  MoveL 4024 to (-41.13, 53.64, 69.25) mm, rotated rx -180 ry 0 rz 180 deg; joints [-165.068, 60.327, -74.122, 164.646, 76.68, 3.62]
  Call Extruder(59.42806)
  MoveL 4025 to (-41.09, 53.05, 69.25) mm, rotated rx -180 ry 0 rz -180 deg; joints [-165.222, 60.313, -74.132, 164.802, 76.647, 3.59]
  MoveL 4026 to (-41.09, 53.05, 69.25) mm, rotated rx -180 ry 0 rz -180 deg; joints [-165.222, 60.313, -74.132, 164.802, 76.647, 3.59]
  Call Extruder(59.67430)
  MoveL 4027 to (-41.04, 52.56, 69.25) mm, rotated rx -180 ry 0 rz -180 deg; joints [-165.349, 60.302, -74.14, 164.93, 76.62, 3.565]
  MoveL 4028 to (-41.04, 52.56, 69.25) mm, rotated rx -180 ry 0 rz -180 deg; joints [-165.349, 60.302, -74.14, 164.93, 76.62, 3.565]
  Call Extruder(59.87100)
  MoveL 4029 to (-40.99, 52.17, 69.25) mm, rotated rx 180 ry 0 rz 180 deg; joints [-165.449, 60.292, -74.147, 165.032, 76.597, 3.546]
  MoveL 4030 to (-40.99, 52.17, 69.25) mm, rotated rx 180 ry 0 rz 180 deg; joints [-165.449, 60.292, -74.147, 165.032, 76.597, 3.546]
  Call Extruder(60.06858)
  MoveL 4031 to (-40.95, 51.78, 69.25) mm, rotated rx -180 ry 0 rz -180 deg; joints [-165.549, 60.282, -74.154, 165.134, 76.575, 3.527]
  MoveL 4032 to (-40.95, 51.78, 69.25) mm, rotated rx -180 ry 0 rz -180 deg; joints [-165.549, 60.282, -74.154, 165.134, 76.575, 3.527]
  Call Extruder(60.26702)
  MoveL 4033 to (-40.9, 51.4, 69.25) mm, rotated rx 180 ry 0 rz -180 deg; joints [-165.65, 60.272, -74.162, 165.236, 76.552, 3.507]
  MoveL 4034 to (-40.9, 51.4, 69.25) mm, rotated rx 180 ry 0 rz -180 deg; joints [-165.65, 60.272, -74.162, 165.236, 76.552, 3.507]
  Call Extruder(60.46633)
  MoveL 4035 to (-40.86, 51.01, 69.25) mm, rotated rx -180 ry 0 rz -180 deg; joints [-165.751, 60.262, -74.169, 165.339, 76.53, 3.488]
  MoveL 4036 to (-40.86, 51.01, 69.25) mm, rotated rx -180 ry 0 rz -180 deg; joints [-165.751, 60.262, -74.169, 165.339, 76.53, 3.488]
  Call Extruder(60.62514)
  MoveL 4037 to (-40.81, 50.7, 69.25) mm, rotated rx 180 ry 0 rz -180 deg; joints [-165.829, 60.254, -74.175, 165.419, 76.511, 3.472]
  MoveL 4038 to (-40.81, 50.7, 69.25) mm, rotated rx 180 ry 0 rz -180 deg; joints [-165.829, 60.254, -74.175, 165.419, 76.511, 3.472]
  Call Extruder(60.78469)
  MoveL 4039 to (-40.76, 50.4, 69.25) mm, rotated rx -180 ry 0 rz -180 deg; joints [-165.908, 60.245, -74.181, 165.499, 76.492, 3.457]
  MoveL 4040 to (-40.76, 50.4, 69.25) mm, rotated rx -180 ry 0 rz -180 deg; joints [-165.908, 60.245, -74.181, 165.499, 76.492, 3.457]
  Call Extruder(60.94496)
  MoveL 4041 to (-40.71, 50.09, 69.25) mm, rotated rx -180 ry 0 rz -180 deg; joints [-165.987, 60.237, -74.187, 165.578, 76.473, 3.442]
  MoveL 4042 to (-40.71, 50.09, 69.25) mm, rotated rx -180 ry 0 rz -180 deg; joints [-165.987, 60.237, -74.187, 165.578, 76.473, 3.442]
  Call Extruder(61.10596)
  MoveL 4043 to (-40.66, 49.79, 69.25) mm, rotated rx 180 ry 0 rz 180 deg; joints [-166.066, 60.228, -74.193, 165.659, 76.454, 3.427]
  MoveL 4044 to (-40.66, 49.79, 69.25) mm, rotated rx 180 ry 0 rz 180 deg; joints [-166.066, 60.228, -74.193, 165.659, 76.454, 3.427]
  Call Extruder(61.26769)
  MoveL 4045 to (-40.61, 49.48, 69.25) mm, rotated rx 180 ry 0 rz 180 deg; joints [-166.145, 60.22, -74.199, 165.739, 76.435, 3.412]
  MoveL 4046 to (-40.61, 49.48, 69.25) mm, rotated rx 180 ry 0 rz 180 deg; joints [-166.145, 60.22, -74.199, 165.739, 76.435, 3.412]
  Call Extruder(61.43014)
  MoveL 4047 to (-40.57, 49.17, 69.25) mm, rotated rx -180 ry 0 rz -180 deg; joints [-166.224, 60.211, -74.205, 165.819, 76.417, 3.396]
  MoveL 4048 to (-40.57, 49.17, 69.25) mm, rotated rx -180 ry 0 rz -180 deg; joints [-166.224, 60.211, -74.205, 165.819, 76.417, 3.396]
  Call Extruder(61.56407)
  MoveL 4049 to (-40.52, 48.93, 69.25) mm, rotated rx -180 ry 0 rz -180 deg; joints [-166.288, 60.204, -74.21, 165.884, 76.4, 3.384]
  MoveL 4050 to (-40.52, 48.93, 69.25) mm, rotated rx -180 ry 0 rz -180 deg; joints [-166.288, 60.204, -74.21, 165.884, 76.4, 3.384]
  Call Extruder(61.69860)
  MoveL 4051 to (-40.47, 48.68, 69.25) mm, rotated rx -180 ry 0 rz 180 deg; joints [-166.352, 60.196, -74.216, 165.949, 76.384, 3.372]
  MoveL 4052 to (-40.47, 48.68, 69.25) mm, rotated rx -180 ry 0 rz 180 deg; joints [-166.352, 60.196, -74.216, 165.949, 76.384, 3.372]
  Call Extruder(61.83375)
  MoveL 4053 to (-40.42, 48.43, 69.25) mm, rotated rx -180 ry 0 rz -180 deg; joints [-166.416, 60.189, -74.221, 166.014, 76.368, 3.359]
  MoveL 4054 to (-40.42, 48.43, 69.25) mm, rotated rx -180 ry 0 rz -180 deg; joints [-166.416, 60.189, -74.221, 166.014, 76.368, 3.359]
  Call Extruder(61.96950)
  MoveL 4055 to (-40.37, 48.18, 69.25) mm, rotated rx -180 ry 0 rz -180 deg; joints [-166.48, 60.181, -74.226, 166.079, 76.352, 3.347]
  MoveL 4056 to (-40.37, 48.18, 69.25) mm, rotated rx -180 ry 0 rz -180 deg; joints [-166.48, 60.181, -74.226, 166.079, 76.352, 3.347]
  Call Extruder(62.10587)
  MoveL 4057 to (-40.32, 47.93, 69.25) mm, rotated rx -180 ry 0 rz 180 deg; joints [-166.544, 60.174, -74.231, 166.144, 76.336, 3.335]
  MoveL 4058 to (-40.32, 47.93, 69.25) mm, rotated rx -180 ry 0 rz 180 deg; joints [-166.544, 60.174, -74.231, 166.144, 76.336, 3.335]
  Call Extruder(62.24285)
  MoveL 4059 to (-40.27, 47.68, 69.25) mm, rotated rx -180 ry 0 rz -180 deg; joints [-166.608, 60.166, -74.237, 166.21, 76.32, 3.322]
  MoveL 4060 to (-40.27, 47.68, 69.25) mm, rotated rx -180 ry 0 rz -180 deg; joints [-166.608, 60.166, -74.237, 166.21, 76.32, 3.322]
  Call Extruder(62.38043)
  MoveL 4061 to (-40.22, 47.43, 69.25) mm, rotated rx -180 ry 0 rz 180 deg; joints [-166.673, 60.159, -74.242, 166.275, 76.304, 3.31]
  MoveL 4062 to (-40.22, 47.43, 69.25) mm, rotated rx -180 ry 0 rz 180 deg; joints [-166.673, 60.159, -74.242, 166.275, 76.304, 3.31]
  Call Extruder(62.49416)
  MoveL 4063 to (-40.17, 47.23, 69.25) mm, rotated rx -180 ry 0 rz 180 deg; joints [-166.725, 60.152, -74.246, 166.328, 76.29, 3.3]
  MoveL 4064 to (-40.17, 47.23, 69.25) mm, rotated rx -180 ry 0 rz 180 deg; joints [-166.725, 60.152, -74.246, 166.328, 76.29, 3.3]
  Call Extruder(62.60834)
  MoveL 4065 to (-40.13, 47.02, 69.25) mm, rotated rx -180 ry 0 rz 180 deg; joints [-166.778, 60.146, -74.251, 166.382, 76.276, 3.289]
  MoveL 4066 to (-40.13, 47.02, 69.25) mm, rotated rx -180 ry 0 rz 180 deg; joints [-166.778, 60.146, -74.251, 166.382, 76.276, 3.289]
  Call Extruder(62.72297)
  MoveL 4067 to (-40.08, 46.82, 69.25) mm, rotated rx 180 ry 0 rz -180 deg; joints [-166.83, 60.14, -74.255, 166.435, 76.263, 3.279]
  MoveL 4068 to (-40.08, 46.82, 69.25) mm, rotated rx 180 ry 0 rz -180 deg; joints [-166.83, 60.14, -74.255, 166.435, 76.263, 3.279]
  Call Extruder(62.83806)
  MoveL 4069 to (-40.04, 46.61, 69.25) mm, rotated rx -180 ry 0 rz -180 deg; joints [-166.883, 60.133, -74.26, 166.489, 76.249, 3.269]
  MoveL 4070 to (-40.04, 46.61, 69.25) mm, rotated rx -180 ry 0 rz -180 deg; joints [-166.883, 60.133, -74.26, 166.489, 76.249, 3.269]
  Call Extruder(62.96029)
  MoveL 4071 to (-39.98, 46.4, 69.25) mm, rotated rx -180 ry 0 rz -180 deg; joints [-166.937, 60.126, -74.265, 166.544, 76.234, 3.259]
  MoveL 4072 to (-39.98, 46.4, 69.25) mm, rotated rx -180 ry 0 rz -180 deg; joints [-166.937, 60.126, -74.265, 166.544, 76.234, 3.259]
  Call Extruder(63.08996)
  MoveL 4073 to (-39.92, 46.18, 69.25) mm, rotated rx -180 ry 0 rz -180 deg; joints [-166.994, 60.118, -74.271, 166.601, 76.218, 3.248]
  MoveL 4074 to (-39.92, 46.18, 69.25) mm, rotated rx -180 ry 0 rz -180 deg; joints [-166.994, 60.118, -74.271, 166.601, 76.218, 3.248]
  Call Extruder(63.22019)
  MoveL 4075 to (-39.85, 45.95, 69.25) mm, rotated rx 180 ry 0 rz -180 deg; joints [-167.051, 60.11, -74.276, 166.659, 76.201, 3.238]
  MoveL 4076 to (-39.85, 45.95, 69.25) mm, rotated rx 180 ry 0 rz -180 deg; joints [-167.051, 60.11, -74.276, 166.659, 76.201, 3.238]
  Call Extruder(63.35098)
  MoveL 4077 to (-39.78, 45.73, 69.25) mm, rotated rx 180 ry 0 rz -180 deg; joints [-167.107, 60.101, -74.282, 166.716, 76.184, 3.227]
  MoveL 4078 to (-39.78, 45.73, 69.25) mm, rotated rx 180 ry 0 rz -180 deg; joints [-167.107, 60.101, -74.282, 166.716, 76.184, 3.227]
  Call Extruder(63.48234)
  MoveL 4079 to (-39.71, 45.5, 69.25) mm, rotated rx -180 ry 0 rz -180 deg; joints [-167.164, 60.093, -74.288, 166.774, 76.167, 3.216]
  MoveL 4080 to (-39.71, 45.5, 69.25) mm, rotated rx -180 ry 0 rz -180 deg; joints [-167.164, 60.093, -74.288, 166.774, 76.167, 3.216]
  Call Extruder(63.59424)
  MoveL 4081 to (-39.65, 45.32, 69.25) mm, rotated rx -180 ry 0 rz -180 deg; joints [-167.212, 60.086, -74.293, 166.822, 76.153, 3.207]
  MoveL 4082 to (-39.65, 45.32, 69.25) mm, rotated rx -180 ry 0 rz -180 deg; joints [-167.212, 60.086, -74.293, 166.822, 76.153, 3.207]
  Call Extruder(63.70659)
  MoveL 4083 to (-39.59, 45.13, 69.25) mm, rotated rx 180 ry 0 rz 180 deg; joints [-167.26, 60.079, -74.298, 166.871, 76.138, 3.198]
  MoveL 4084 to (-39.59, 45.13, 69.25) mm, rotated rx 180 ry 0 rz 180 deg; joints [-167.26, 60.079, -74.298, 166.871, 76.138, 3.198]
  Call Extruder(63.81938)
  MoveL 4085 to (-39.53, 44.94, 69.25) mm, rotated rx -180 ry 0 rz 180 deg; joints [-167.307, 60.072, -74.303, 166.919, 76.124, 3.19]
  MoveL 4086 to (-39.53, 44.94, 69.25) mm, rotated rx -180 ry 0 rz 180 deg; joints [-167.307, 60.072, -74.303, 166.919, 76.124, 3.19]
  Call Extruder(63.93261)
  MoveL 4087 to (-39.47, 44.75, 69.25) mm, rotated rx -180 ry 0 rz -180 deg; joints [-167.355, 60.065, -74.308, 166.967, 76.109, 3.181]
  MoveL 4088 to (-39.47, 44.75, 69.25) mm, rotated rx -180 ry 0 rz -180 deg; joints [-167.355, 60.065, -74.308, 166.967, 76.109, 3.181]
  Call Extruder(64.04629)
  MoveL 4089 to (-39.41, 44.56, 69.25) mm, rotated rx -180 ry 0 rz -180 deg; joints [-167.403, 60.057, -74.313, 167.016, 76.095, 3.172]
  MoveL 4090 to (-39.41, 44.56, 69.25) mm, rotated rx -180 ry 0 rz -180 deg; joints [-167.403, 60.057, -74.313, 167.016, 76.095, 3.172]
  Call Extruder(64.22825)
  MoveL 4091 to (-39.29, 44.27, 69.25) mm, rotated rx -180 ry 0 rz 180 deg; joints [-167.475, 60.045, -74.321, 167.089, 76.07, 3.159]
  MoveL 4092 to (-39.29, 44.27, 69.25) mm, rotated rx -180 ry 0 rz 180 deg; joints [-167.475, 60.045, -74.321, 167.089, 76.07, 3.159]
  Call Extruder(64.41097)
  MoveL 4093 to (-39.17, 43.98, 69.25) mm, rotated rx 180 ry 0 rz 180 deg; joints [-167.548, 60.032, -74.33, 167.163, 76.045, 3.146]
  MoveL 4094 to (-39.17, 43.98, 69.25) mm, rotated rx 180 ry 0 rz 180 deg; joints [-167.548, 60.032, -74.33, 167.163, 76.045, 3.146]
  Call Extruder(64.58138)
  MoveL 4095 to (-39.05, 43.71, 69.25) mm, rotated rx -180 ry 0 rz -180 deg; joints [-167.615, 60.02, -74.339, 167.231, 76.021, 3.134]
  MoveL 4096 to (-39.05, 43.71, 69.25) mm, rotated rx -180 ry 0 rz -180 deg; joints [-167.615, 60.02, -74.339, 167.231, 76.021, 3.134]
  Call Extruder(64.73937)
  MoveL 4097 to (-38.94, 43.46, 69.25) mm, rotated rx -180 ry 0 rz 180 deg; joints [-167.677, 60.008, -74.346, 167.294, 75.999, 3.122]
  MoveL 4098 to (-38.94, 43.46, 69.25) mm, rotated rx -180 ry 0 rz 180 deg; joints [-167.677, 60.008, -74.346, 167.294, 75.999, 3.122]
  Call Extruder(64.89795)
  MoveL 4099 to (-38.84, 43.21, 69.25) mm, rotated rx -180 ry 0 rz -180 deg; joints [-167.739, 59.997, -74.354, 167.357, 75.977, 3.111]
  MoveL 4100 to (-38.84, 43.21, 69.25) mm, rotated rx -180 ry 0 rz -180 deg; joints [-167.739, 59.997, -74.354, 167.357, 75.977, 3.111]
  Call Extruder(65.10412)
  MoveL 4101 to (-38.66, 42.91, 69.25) mm, rotated rx -180 ry 0 rz -180 deg; joints [-167.813, 59.981, -74.365, 167.431, 75.946, 3.099]
  MoveL 4102 to (-38.66, 42.91, 69.25) mm, rotated rx -180 ry 0 rz -180 deg; joints [-167.813, 59.981, -74.365, 167.431, 75.946, 3.099]
  Call Extruder(65.31106)
  MoveL 4103 to (-38.49, 42.6, 69.25) mm, rotated rx -180 ry 0 rz 180 deg; joints [-167.886, 59.964, -74.377, 167.505, 75.914, 3.087]
  MoveL 4104 to (-38.49, 42.6, 69.25) mm, rotated rx -180 ry 0 rz 180 deg; joints [-167.886, 59.964, -74.377, 167.505, 75.914, 3.087]
  Call Extruder(65.51879)
  MoveL 4105 to (-38.31, 42.3, 69.25) mm, rotated rx 180 ry 0 rz 180 deg; joints [-167.96, 59.947, -74.388, 167.579, 75.883, 3.075]
  MoveL 4106 to (-38.31, 42.3, 69.25) mm, rotated rx 180 ry 0 rz 180 deg; joints [-167.96, 59.947, -74.388, 167.579, 75.883, 3.075]
  Call Extruder(65.72729)
  MoveL 4107 to (-38.14, 41.99, 69.25) mm, rotated rx -180 ry 0 rz -180 deg; joints [-168.033, 59.93, -74.4, 167.653, 75.852, 3.063]
  MoveL 4108 to (-38.14, 41.99, 69.25) mm, rotated rx -180 ry 0 rz -180 deg; joints [-168.033, 59.93, -74.4, 167.653, 75.852, 3.063]
  Call Extruder(65.90684)
  MoveL 4109 to (-37.96, 41.75, 69.25) mm, rotated rx 180 ry 0 rz -180 deg; joints [-168.091, 59.914, -74.41, 167.711, 75.822, 3.054]
  MoveL 4110 to (-37.96, 41.75, 69.25) mm, rotated rx 180 ry 0 rz -180 deg; joints [-168.091, 59.914, -74.41, 167.711, 75.822, 3.054]
  Call Extruder(66.24028)
  MoveL 4111 to (-37.63, 41.3, 69.25) mm, rotated rx -180 ry 0 rz -180 deg; joints [-168.197, 59.885, -74.43, 167.818, 75.768, 3.038]
  MoveL 4112 to (-37.63, 41.3, 69.25) mm, rotated rx -180 ry 0 rz -180 deg; joints [-168.197, 59.885, -74.43, 167.818, 75.768, 3.038]
  Call Extruder(66.57490)
  MoveL 4113 to (-37.3, 40.85, 69.25) mm, rotated rx 180 ry 0 rz -180 deg; joints [-168.304, 59.855, -74.45, 167.925, 75.714, 3.022]
  Call Extruder(67.40283)
  MoveL 4114 to (-36.39, 39.81, 69.25) mm, rotated rx 180 ry 0 rz 180 deg; joints [-168.541, 59.776, -74.503, 168.163, 75.573, 2.989]
  Call Extruder(68.23074)
  MoveL 4115 to (-35.35, 38.9, 69.25) mm, rotated rx -180 ry 0 rz 180 deg; joints [-168.739, 59.69, -74.559, 168.359, 75.423, 2.968]
  Call Extruder(68.39804)
  MoveL 4116 to (-35.13, 38.73, 69.25) mm, rotated rx -180 ry 0 rz 180 deg; joints [-168.773, 59.671, -74.571, 168.392, 75.392, 2.966]
  MoveL 4117 to (-35.13, 38.73, 69.25) mm, rotated rx -180 ry 0 rz 180 deg; joints [-168.773, 59.671, -74.571, 168.392, 75.392, 2.966]
  Call Extruder(68.73147)
  MoveL 4118 to (-34.68, 38.41, 69.25) mm, rotated rx -180 ry 0 rz 180 deg; joints [-168.84, 59.635, -74.595, 168.459, 75.329, 2.961]
  MoveL 4119 to (-34.68, 38.41, 69.25) mm, rotated rx -180 ry 0 rz 180 deg; joints [-168.84, 59.635, -74.595, 168.459, 75.329, 2.961]
  Call Extruder(69.06371)
  MoveL 4120 to (-34.23, 38.08, 69.25) mm, rotated rx 180 ry 0 rz -180 deg; joints [-168.908, 59.598, -74.619, 168.526, 75.266, 2.955]
  MoveL 4121 to (-34.23, 38.08, 69.25) mm, rotated rx 180 ry 0 rz -180 deg; joints [-168.908, 59.598, -74.619, 168.526, 75.266, 2.955]
  Call Extruder(69.18141)
  MoveL 4122 to (-34.05, 37.98, 69.25) mm, rotated rx -180 ry 0 rz 180 deg; joints [-168.927, 59.584, -74.627, 168.544, 75.243, 2.955]
  MoveL 4123 to (-34.05, 37.98, 69.25) mm, rotated rx -180 ry 0 rz 180 deg; joints [-168.927, 59.584, -74.627, 168.544, 75.243, 2.955]
  Call Extruder(69.38913)
  MoveL 4124 to (-33.75, 37.8, 69.25) mm, rotated rx -180 ry 0 rz 180 deg; joints [-168.96, 59.56, -74.643, 168.576, 75.203, 2.954]
  MoveL 4125 to (-33.75, 37.8, 69.25) mm, rotated rx -180 ry 0 rz 180 deg; joints [-168.96, 59.56, -74.643, 168.576, 75.203, 2.954]
  Call Extruder(69.59607)
  MoveL 4126 to (-33.45, 37.63, 69.25) mm, rotated rx -180 ry 0 rz 180 deg; joints [-168.993, 59.536, -74.658, 168.609, 75.162, 2.954]
  MoveL 4127 to (-33.45, 37.63, 69.25) mm, rotated rx -180 ry 0 rz 180 deg; joints [-168.993, 59.536, -74.658, 168.609, 75.162, 2.954]
  Call Extruder(69.80224)
  MoveL 4128 to (-33.14, 37.45, 69.25) mm, rotated rx -180 ry 0 rz -180 deg; joints [-169.026, 59.512, -74.673, 168.641, 75.122, 2.953]
  MoveL 4129 to (-33.14, 37.45, 69.25) mm, rotated rx -180 ry 0 rz -180 deg; joints [-169.026, 59.512, -74.673, 168.641, 75.122, 2.953]
  Call Extruder(69.98392)
  MoveL 4130 to (-32.86, 37.31, 69.25) mm, rotated rx 180 ry 0 rz 180 deg; joints [-169.052, 59.49, -74.687, 168.665, 75.086, 2.953]
  MoveL 4131 to (-32.86, 37.31, 69.25) mm, rotated rx 180 ry 0 rz 180 deg; joints [-169.052, 59.49, -74.687, 168.665, 75.086, 2.953]
  Call Extruder(70.14192)
  MoveL 4132 to (-32.62, 37.2, 69.25) mm, rotated rx -180 ry 0 rz -180 deg; joints [-169.068, 59.47, -74.699, 168.681, 75.054, 2.955]
  MoveL 4133 to (-32.62, 37.2, 69.25) mm, rotated rx -180 ry 0 rz -180 deg; joints [-169.068, 59.47, -74.699, 168.681, 75.054, 2.955]
  Call Extruder(70.29931)
  MoveL 4134 to (-32.37, 37.1, 69.25) mm, rotated rx 180 ry 0 rz -180 deg; joints [-169.085, 59.451, -74.711, 168.697, 75.022, 2.957]
  MoveL 4135 to (-32.37, 37.1, 69.25) mm, rotated rx 180 ry 0 rz -180 deg; joints [-169.085, 59.451, -74.711, 168.697, 75.022, 2.957]
  Call Extruder(70.48203)
  MoveL 4136 to (-32.07, 36.97, 69.25) mm, rotated rx 180 ry 0 rz 180 deg; joints [-169.104, 59.428, -74.726, 168.714, 74.985, 2.96]
  MoveL 4137 to (-32.07, 36.97, 69.25) mm, rotated rx 180 ry 0 rz 180 deg; joints [-169.104, 59.428, -74.726, 168.714, 74.985, 2.96]
  Call Extruder(70.66398)
  MoveL 4138 to (-31.78, 36.85, 69.25) mm, rotated rx -180 ry 0 rz 180 deg; joints [-169.122, 59.406, -74.74, 168.731, 74.948, 2.962]
  MoveL 4139 to (-31.78, 36.85, 69.25) mm, rotated rx -180 ry 0 rz 180 deg; joints [-169.122, 59.406, -74.74, 168.731, 74.948, 2.962]
  Call Extruder(70.81131)
  MoveL 4140 to (-31.54, 36.76, 69.25) mm, rotated rx -180 ry 0 rz -180 deg; joints [-169.135, 59.387, -74.751, 168.743, 74.918, 2.965]
  MoveL 4141 to (-31.54, 36.76, 69.25) mm, rotated rx -180 ry 0 rz -180 deg; joints [-169.135, 59.387, -74.751, 168.743, 74.918, 2.965]
  Call Extruder(70.92455)
  MoveL 4142 to (-31.35, 36.7, 69.25) mm, rotated rx 180 ry 0 rz 180 deg; joints [-169.143, 59.373, -74.76, 168.749, 74.894, 2.968]
  MoveL 4143 to (-31.35, 36.7, 69.25) mm, rotated rx 180 ry 0 rz 180 deg; joints [-169.143, 59.373, -74.76, 168.749, 74.894, 2.968]
  Call Extruder(71.03734)
  MoveL 4144 to (-31.17, 36.64, 69.25) mm, rotated rx -180 ry 0 rz -180 deg; joints [-169.15, 59.358, -74.769, 168.755, 74.871, 2.97]
  MoveL 4145 to (-31.17, 36.64, 69.25) mm, rotated rx -180 ry 0 rz -180 deg; joints [-169.15, 59.358, -74.769, 168.755, 74.871, 2.97]
  Call Extruder(71.14968)
  MoveL 4146 to (-30.98, 36.58, 69.25) mm, rotated rx 180 ry 0 rz 180 deg; joints [-169.157, 59.344, -74.778, 168.762, 74.848, 2.973]
  MoveL 4147 to (-30.98, 36.58, 69.25) mm, rotated rx 180 ry 0 rz 180 deg; joints [-169.157, 59.344, -74.778, 168.762, 74.848, 2.973]
  Call Extruder(71.26159)
  MoveL 4148 to (-30.79, 36.52, 69.25) mm, rotated rx -180 ry 0 rz -180 deg; joints [-169.164, 59.329, -74.787, 168.768, 74.825, 2.976]
  MoveL 4149 to (-30.79, 36.52, 69.25) mm, rotated rx -180 ry 0 rz -180 deg; joints [-169.164, 59.329, -74.787, 168.768, 74.825, 2.976]
  Call Extruder(71.38299)
  MoveL 4150 to (-30.58, 36.45, 69.25) mm, rotated rx -180 ry 0 rz -180 deg; joints [-169.172, 59.313, -74.797, 168.774, 74.799, 2.979]
  MoveL 4151 to (-30.58, 36.45, 69.25) mm, rotated rx -180 ry 0 rz -180 deg; joints [-169.172, 59.313, -74.797, 168.774, 74.799, 2.979]
  Call Extruder(71.51378)
  MoveL 4152 to (-30.36, 36.38, 69.25) mm, rotated rx -180 ry 0 rz 180 deg; joints [-169.179, 59.296, -74.807, 168.78, 74.772, 2.983]
  MoveL 4153 to (-30.36, 36.38, 69.25) mm, rotated rx -180 ry 0 rz 180 deg; joints [-169.179, 59.296, -74.807, 168.78, 74.772, 2.983]
  Call Extruder(71.64400)
  MoveL 4154 to (-30.14, 36.32, 69.25) mm, rotated rx 180 ry 0 rz 180 deg; joints [-169.186, 59.279, -74.817, 168.786, 74.744, 2.986]
  MoveL 4155 to (-30.14, 36.32, 69.25) mm, rotated rx 180 ry 0 rz 180 deg; joints [-169.186, 59.279, -74.817, 168.786, 74.744, 2.986]
  Call Extruder(71.77367)
  MoveL 4156 to (-29.91, 36.25, 69.25) mm, rotated rx -180 ry 0 rz 180 deg; joints [-169.193, 59.262, -74.828, 168.792, 74.717, 2.99]
  MoveL 4157 to (-29.91, 36.25, 69.25) mm, rotated rx -180 ry 0 rz 180 deg; joints [-169.193, 59.262, -74.828, 168.792, 74.717, 2.99]
  Call Extruder(71.90276)
  MoveL 4158 to (-29.69, 36.18, 69.25) mm, rotated rx -180 ry 0 rz -180 deg; joints [-169.201, 59.245, -74.838, 168.798, 74.689, 2.993]
  MoveL 4159 to (-29.69, 36.18, 69.25) mm, rotated rx -180 ry 0 rz -180 deg; joints [-169.201, 59.245, -74.838, 168.798, 74.689, 2.993]
  Call Extruder(72.01784)
  MoveL 4160 to (-29.48, 36.14, 69.25) mm, rotated rx -180 ry 0 rz 180 deg; joints [-169.202, 59.229, -74.848, 168.799, 74.665, 2.998]
  MoveL 4161 to (-29.48, 36.14, 69.25) mm, rotated rx -180 ry 0 rz 180 deg; joints [-169.202, 59.229, -74.848, 168.799, 74.665, 2.998]
  Call Extruder(72.13246)
  MoveL 4162 to (-29.28, 36.09, 69.25) mm, rotated rx -180 ry 0 rz -180 deg; joints [-169.204, 59.214, -74.857, 168.799, 74.64, 3.002]
  MoveL 4163 to (-29.28, 36.09, 69.25) mm, rotated rx -180 ry 0 rz -180 deg; joints [-169.204, 59.214, -74.857, 168.799, 74.64, 3.002]
  Call Extruder(72.24663)
  MoveL 4164 to (-29.08, 36.05, 69.25) mm, rotated rx 180 ry 0 rz 180 deg; joints [-169.206, 59.198, -74.866, 168.799, 74.616, 3.007]
  MoveL 4165 to (-29.08, 36.05, 69.25) mm, rotated rx 180 ry 0 rz 180 deg; joints [-169.206, 59.198, -74.866, 168.799, 74.616, 3.007]
  Call Extruder(72.36034)
  MoveL 4166 to (-28.87, 36, 69.25) mm, rotated rx 180 ry 0 rz 180 deg; joints [-169.207, 59.183, -74.876, 168.8, 74.591, 3.012]
  MoveL 4167 to (-28.87, 36, 69.25) mm, rotated rx 180 ry 0 rz 180 deg; joints [-169.207, 59.183, -74.876, 168.8, 74.591, 3.012]
  Call Extruder(72.48576)
  MoveL 4168 to (-28.65, 35.96, 69.25) mm, rotated rx -180 ry 0 rz -180 deg; joints [-169.208, 59.165, -74.886, 168.8, 74.565, 3.017]
  MoveL 4169 to (-28.65, 35.96, 69.25) mm, rotated rx -180 ry 0 rz -180 deg; joints [-169.208, 59.165, -74.886, 168.8, 74.565, 3.017]
  Call Extruder(72.62274)
  MoveL 4170 to (-28.4, 35.91, 69.25) mm, rotated rx -180 ry 0 rz 180 deg; joints [-169.209, 59.146, -74.897, 168.799, 74.535, 3.023]
  MoveL 4171 to (-28.4, 35.91, 69.25) mm, rotated rx -180 ry 0 rz 180 deg; joints [-169.209, 59.146, -74.897, 168.799, 74.535, 3.023]
  Call Extruder(72.75911)
  MoveL 4172 to (-28.15, 35.86, 69.25) mm, rotated rx 180 ry 0 rz -180 deg; joints [-169.21, 59.128, -74.908, 168.797, 74.505, 3.029]
  MoveL 4173 to (-28.15, 35.86, 69.25) mm, rotated rx 180 ry 0 rz -180 deg; joints [-169.21, 59.128, -74.908, 168.797, 74.505, 3.029]
  Call Extruder(72.89487)
  MoveL 4174 to (-27.9, 35.81, 69.25) mm, rotated rx -180 ry 0 rz 180 deg; joints [-169.21, 59.109, -74.92, 168.797, 74.476, 3.035]
  MoveL 4175 to (-27.9, 35.81, 69.25) mm, rotated rx -180 ry 0 rz 180 deg; joints [-169.21, 59.109, -74.92, 168.797, 74.476, 3.035]
  Call Extruder(73.03001)
  MoveL 4176 to (-27.65, 35.76, 69.25) mm, rotated rx -180 ry 0 rz 180 deg; joints [-169.211, 59.09, -74.931, 168.795, 74.446, 3.04]
  MoveL 4177 to (-27.65, 35.76, 69.25) mm, rotated rx -180 ry 0 rz 180 deg; joints [-169.211, 59.09, -74.931, 168.795, 74.446, 3.04]
  Call Extruder(73.16455)
  MoveL 4178 to (-27.4, 35.71, 69.25) mm, rotated rx 180 ry 0 rz -180 deg; joints [-169.212, 59.071, -74.942, 168.795, 74.417, 3.046]
  MoveL 4179 to (-27.4, 35.71, 69.25) mm, rotated rx 180 ry 0 rz -180 deg; joints [-169.212, 59.071, -74.942, 168.795, 74.417, 3.046]
  Call Extruder(73.29848)
  MoveL 4180 to (-27.15, 35.66, 69.25) mm, rotated rx 180 ry 0 rz 180 deg; joints [-169.212, 59.052, -74.953, 168.793, 74.387, 3.052]
  MoveL 4181 to (-27.15, 35.66, 69.25) mm, rotated rx 180 ry 0 rz 180 deg; joints [-169.212, 59.052, -74.953, 168.793, 74.387, 3.052]
  Call Extruder(73.44634)
  MoveL 4182 to (-26.87, 35.61, 69.25) mm, rotated rx -180 ry 0 rz 180 deg; joints [-169.211, 59.031, -74.965, 168.791, 74.354, 3.059]
  MoveL 4183 to (-26.87, 35.61, 69.25) mm, rotated rx -180 ry 0 rz 180 deg; joints [-169.211, 59.031, -74.965, 168.791, 74.354, 3.059]
  Call Extruder(73.60807)
  MoveL 4184 to (-26.57, 35.56, 69.25) mm, rotated rx -180 ry 0 rz -180 deg; joints [-169.208, 59.007, -74.979, 168.786, 74.318, 3.068]
  MoveL 4185 to (-26.57, 35.56, 69.25) mm, rotated rx -180 ry 0 rz -180 deg; joints [-169.208, 59.007, -74.979, 168.786, 74.318, 3.068]
  Call Extruder(73.76908)
  MoveL 4186 to (-26.26, 35.51, 69.25) mm, rotated rx 180 ry 0 rz 180 deg; joints [-169.205, 58.984, -74.992, 168.78, 74.283, 3.076]
  MoveL 4187 to (-26.26, 35.51, 69.25) mm, rotated rx 180 ry 0 rz 180 deg; joints [-169.205, 58.984, -74.992, 168.78, 74.283, 3.076]
  Call Extruder(73.92935)
  MoveL 4188 to (-25.96, 35.47, 69.25) mm, rotated rx -180 ry 0 rz -180 deg; joints [-169.202, 58.961, -75.006, 168.776, 74.247, 3.084]
  MoveL 4189 to (-25.96, 35.47, 69.25) mm, rotated rx -180 ry 0 rz -180 deg; joints [-169.202, 58.961, -75.006, 168.776, 74.247, 3.084]
  Call Extruder(74.08890)
  MoveL 4190 to (-25.65, 35.42, 69.25) mm, rotated rx -180 ry 0 rz 180 deg; joints [-169.199, 58.938, -75.019, 168.77, 74.211, 3.092]
  MoveL 4191 to (-25.65, 35.42, 69.25) mm, rotated rx -180 ry 0 rz 180 deg; joints [-169.199, 58.938, -75.019, 168.77, 74.211, 3.092]
  Call Extruder(74.24773)
  MoveL 4192 to (-25.34, 35.37, 69.25) mm, rotated rx -180 ry 0 rz 180 deg; joints [-169.196, 58.914, -75.032, 168.765, 74.175, 3.1]
  MoveL 4193 to (-25.34, 35.37, 69.25) mm, rotated rx -180 ry 0 rz 180 deg; joints [-169.196, 58.914, -75.032, 168.765, 74.175, 3.1]
  Call Extruder(74.42640)
  MoveL 4194 to (-25, 35.32, 69.25) mm, rotated rx 180 ry 0 rz 180 deg; joints [-169.191, 58.888, -75.047, 168.757, 74.135, 3.11]
  MoveL 4195 to (-25, 35.32, 69.25) mm, rotated rx 180 ry 0 rz 180 deg; joints [-169.191, 58.888, -75.047, 168.757, 74.135, 3.11]
  Call Extruder(74.62484)
  MoveL 4196 to (-24.61, 35.28, 69.25) mm, rotated rx -180 ry 0 rz 180 deg; joints [-169.182, 58.859, -75.064, 168.746, 74.09, 3.122]
  MoveL 4197 to (-24.61, 35.28, 69.25) mm, rotated rx -180 ry 0 rz 180 deg; joints [-169.182, 58.859, -75.064, 168.746, 74.09, 3.122]
  Call Extruder(74.82241)
  MoveL 4198 to (-24.22, 35.23, 69.25) mm, rotated rx 180 ry 0 rz 180 deg; joints [-169.174, 58.829, -75.081, 168.735, 74.046, 3.134]
  MoveL 4199 to (-24.22, 35.23, 69.25) mm, rotated rx 180 ry 0 rz 180 deg; joints [-169.174, 58.829, -75.081, 168.735, 74.046, 3.134]
  Call Extruder(75.01912)
  MoveL 4200 to (-23.83, 35.18, 69.25) mm, rotated rx -180 ry 0 rz -180 deg; joints [-169.166, 58.8, -75.097, 168.723, 74.001, 3.146]
  MoveL 4201 to (-23.83, 35.18, 69.25) mm, rotated rx -180 ry 0 rz -180 deg; joints [-169.166, 58.8, -75.097, 168.723, 74.001, 3.146]
  Call Extruder(75.21496)
  MoveL 4202 to (-23.45, 35.14, 69.25) mm, rotated rx 180 ry 0 rz -180 deg; joints [-169.157, 58.77, -75.114, 168.712, 73.956, 3.158]
  MoveL 4203 to (-23.45, 35.14, 69.25) mm, rotated rx 180 ry 0 rz -180 deg; joints [-169.157, 58.77, -75.114, 168.712, 73.956, 3.158]
  Call Extruder(75.51035)
  MoveL 4204 to (-22.86, 35.09, 69.25) mm, rotated rx -180 ry 0 rz 180 deg; joints [-169.137, 58.726, -75.139, 168.687, 73.889, 3.177]
  MoveL 4205 to (-22.86, 35.09, 69.25) mm, rotated rx -180 ry 0 rz 180 deg; joints [-169.137, 58.726, -75.139, 168.687, 73.889, 3.177]
  Call Extruder(75.80442)
  MoveL 4206 to (-22.27, 35.04, 69.25) mm, rotated rx 180 ry 0 rz 180 deg; joints [-169.117, 58.681, -75.163, 168.662, 73.823, 3.198]
  MoveL 4207 to (-22.27, 35.04, 69.25) mm, rotated rx 180 ry 0 rz 180 deg; joints [-169.117, 58.681, -75.163, 168.662, 73.823, 3.198]
  Call Extruder(76.09715)
  MoveL 4208 to (-21.68, 35, 69.25) mm, rotated rx -180 ry 0 rz 180 deg; joints [-169.096, 58.636, -75.188, 168.637, 73.756, 3.218]
  MoveL 4209 to (-21.68, 35, 69.25) mm, rotated rx -180 ry 0 rz 180 deg; joints [-169.096, 58.636, -75.188, 168.637, 73.756, 3.218]
  Call Extruder(76.67060)
  MoveL 4210 to (-20.52, 34.95, 69.25) mm, rotated rx -180 ry 0 rz -180 deg; joints [-169.042, 58.548, -75.235, 168.573, 73.626, 3.261]
  MoveL 4211 to (-20.52, 34.95, 69.25) mm, rotated rx -180 ry 0 rz -180 deg; joints [-169.042, 58.548, -75.235, 168.573, 73.626, 3.261]
  Call Extruder(77.38456)
  MoveL 4212 to (-19.06, 34.91, 69.25) mm, rotated rx -180 ry 0 rz 180 deg; joints [-168.967, 58.438, -75.294, 168.485, 73.464, 3.318]
  Call Extruder(194.23128)
  MoveL 4213 to (219.06, 34.91, 69.25) mm, rotated rx 180 ry 0 rz 180 deg; joints [-30.588, 47.996, -77.471, 34.176, 115.06, 16.045]
  Call Extruder(194.65984)
  MoveL 4214 to (219.94, 34.93, 69.25) mm, rotated rx 180 ry 0 rz 180 deg; joints [-30.233, 48.077, -77.472, 33.779, 115.092, 15.837]
  MoveL 4215 to (219.94, 34.93, 69.25) mm, rotated rx 180 ry 0 rz 180 deg; joints [-30.233, 48.077, -77.472, 33.779, 115.092, 15.837]
  Call Extruder(195.23329)
  MoveL 4216 to (221.1, 34.97, 69.25) mm, rotated rx -180 ry 0 rz 180 deg; joints [-29.789, 48.184, -77.474, 33.279, 115.124, 15.572]
  MoveL 4217 to (221.1, 34.97, 69.25) mm, rotated rx -180 ry 0 rz 180 deg; joints [-29.789, 48.184, -77.474, 33.279, 115.124, 15.572]
  Call Extruder(195.66760)
  MoveL 4218 to (221.97, 35.02, 69.25) mm, rotated rx 180 ry 0 rz 180 deg; joints [-29.47, 48.266, -77.476, 32.92, 115.142, 15.379]
  MoveL 4219 to (221.97, 35.02, 69.25) mm, rotated rx 180 ry 0 rz 180 deg; joints [-29.47, 48.266, -77.476, 32.92, 115.142, 15.379]
  Call Extruder(195.96166)
  MoveL 4220 to (222.56, 35.07, 69.25) mm, rotated rx -180 ry 0 rz 180 deg; joints [-29.272, 48.322, -77.476, 32.694, 115.148, 15.256]
  MoveL 4221 to (222.56, 35.07, 69.25) mm, rotated rx -180 ry 0 rz 180 deg; joints [-29.272, 48.322, -77.476, 32.694, 115.148, 15.256]
  Call Extruder(196.25705)
  MoveL 4222 to (223.15, 35.11, 69.25) mm, rotated rx -180 ry 0 rz -180 deg; joints [-29.075, 48.378, -77.477, 32.47, 115.153, 15.134]
  MoveL 4223 to (223.15, 35.11, 69.25) mm, rotated rx -180 ry 0 rz -180 deg; joints [-29.075, 48.378, -77.477, 32.47, 115.153, 15.134]
  Call Extruder(196.50328)
  MoveL 4224 to (223.64, 35.16, 69.25) mm, rotated rx -180 ry 0 rz 180 deg; joints [-28.92, 48.425, -77.477, 32.293, 115.154, 15.036]
  MoveL 4225 to (223.64, 35.16, 69.25) mm, rotated rx -180 ry 0 rz 180 deg; joints [-28.92, 48.425, -77.477, 32.293, 115.154, 15.036]
  Call Extruder(196.69999)
  MoveL 4226 to (224.03, 35.21, 69.25) mm, rotated rx -180 ry 0 rz 180 deg; joints [-28.804, 48.463, -77.478, 32.16, 115.152, 14.962]
  MoveL 4227 to (224.03, 35.21, 69.25) mm, rotated rx -180 ry 0 rz 180 deg; joints [-28.804, 48.463, -77.478, 32.16, 115.152, 14.962]
  Call Extruder(196.89757)
  MoveL 4228 to (224.42, 35.25, 69.25) mm, rotated rx 180 ry 0 rz 180 deg; joints [-28.69, 48.501, -77.478, 32.029, 115.15, 14.888]
  MoveL 4229 to (224.42, 35.25, 69.25) mm, rotated rx 180 ry 0 rz 180 deg; joints [-28.69, 48.501, -77.478, 32.029, 115.15, 14.888]
  Call Extruder(197.09601)
  MoveL 4230 to (224.8, 35.3, 69.25) mm, rotated rx -180 ry 0 rz 180 deg; joints [-28.577, 48.538, -77.478, 31.899, 115.147, 14.815]
  MoveL 4231 to (224.8, 35.3, 69.25) mm, rotated rx -180 ry 0 rz 180 deg; joints [-28.577, 48.538, -77.478, 31.899, 115.147, 14.815]
  Call Extruder(197.29532)
  MoveL 4232 to (225.19, 35.34, 69.25) mm, rotated rx -180 ry 0 rz 180 deg; joints [-28.465, 48.576, -77.478, 31.77, 115.144, 14.742]
  MoveL 4233 to (225.19, 35.34, 69.25) mm, rotated rx -180 ry 0 rz 180 deg; joints [-28.465, 48.576, -77.478, 31.77, 115.144, 14.742]
  Call Extruder(197.45414)
  MoveL 4234 to (225.5, 35.39, 69.25) mm, rotated rx -180 ry 0 rz 180 deg; joints [-28.385, 48.606, -77.478, 31.677, 115.138, 14.688]
  MoveL 4235 to (225.5, 35.39, 69.25) mm, rotated rx -180 ry 0 rz 180 deg; joints [-28.385, 48.606, -77.478, 31.677, 115.138, 14.688]
  Call Extruder(197.61369)
  MoveL 4236 to (225.8, 35.44, 69.25) mm, rotated rx 180 ry 0 rz 180 deg; joints [-28.307, 48.637, -77.478, 31.586, 115.132, 14.635]
  MoveL 4237 to (225.8, 35.44, 69.25) mm, rotated rx 180 ry 0 rz 180 deg; joints [-28.307, 48.637, -77.478, 31.586, 115.132, 14.635]
  Call Extruder(197.77397)
  MoveL 4238 to (226.11, 35.49, 69.25) mm, rotated rx 180 ry 0 rz 180 deg; joints [-28.228, 48.667, -77.478, 31.495, 115.126, 14.582]
  MoveL 4239 to (226.11, 35.49, 69.25) mm, rotated rx 180 ry 0 rz 180 deg; joints [-28.228, 48.667, -77.478, 31.495, 115.126, 14.582]
  Call Extruder(197.93497)
  MoveL 4240 to (226.41, 35.54, 69.25) mm, rotated rx -180 ry 0 rz 180 deg; joints [-28.151, 48.697, -77.478, 31.405, 115.12, 14.53]
  MoveL 4241 to (226.41, 35.54, 69.25) mm, rotated rx -180 ry 0 rz 180 deg; joints [-28.151, 48.697, -77.478, 31.405, 115.12, 14.53]
  Call Extruder(198.09670)
  MoveL 4242 to (226.72, 35.59, 69.25) mm, rotated rx -180 ry 0 rz 180 deg; joints [-28.074, 48.727, -77.478, 31.315, 115.113, 14.477]
  MoveL 4243 to (226.72, 35.59, 69.25) mm, rotated rx -180 ry 0 rz 180 deg; joints [-28.074, 48.727, -77.478, 31.315, 115.113, 14.477]
  Call Extruder(198.25916)
  MoveL 4244 to (227.02, 35.63, 69.25) mm, rotated rx -180 ry 0 rz 180 deg; joints [-27.998, 48.758, -77.478, 31.226, 115.106, 14.425]
  MoveL 4245 to (227.02, 35.63, 69.25) mm, rotated rx -180 ry 0 rz 180 deg; joints [-27.998, 48.758, -77.478, 31.226, 115.106, 14.425]
  Call Extruder(198.39309)
  MoveL 4246 to (227.27, 35.68, 69.25) mm, rotated rx -180 ry 0 rz 180 deg; joints [-27.942, 48.783, -77.478, 31.161, 115.098, 14.386]
  MoveL 4247 to (227.27, 35.68, 69.25) mm, rotated rx -180 ry 0 rz 180 deg; joints [-27.942, 48.783, -77.478, 31.161, 115.098, 14.386]
  Call Extruder(198.52763)
  MoveL 4248 to (227.52, 35.73, 69.25) mm, rotated rx -180 ry 0 rz 180 deg; joints [-27.888, 48.808, -77.478, 31.096, 115.09, 14.347]
  MoveL 4249 to (227.52, 35.73, 69.25) mm, rotated rx -180 ry 0 rz 180 deg; joints [-27.888, 48.808, -77.478, 31.096, 115.09, 14.347]
  Call Extruder(198.66277)
  MoveL 4250 to (227.77, 35.78, 69.25) mm, rotated rx -180 ry 0 rz 180 deg; joints [-27.834, 48.833, -77.478, 31.032, 115.082, 14.308]
  MoveL 4251 to (227.77, 35.78, 69.25) mm, rotated rx -180 ry 0 rz 180 deg; joints [-27.834, 48.833, -77.478, 31.032, 115.082, 14.308]
  Call Extruder(198.79853)
  MoveL 4252 to (228.02, 35.83, 69.25) mm, rotated rx -180 ry 0 rz 180 deg; joints [-27.78, 48.858, -77.478, 30.968, 115.074, 14.269]
  MoveL 4253 to (228.02, 35.83, 69.25) mm, rotated rx -180 ry 0 rz 180 deg; joints [-27.78, 48.858, -77.478, 30.968, 115.074, 14.269]
  Call Extruder(198.93490)
  MoveL 4254 to (228.27, 35.88, 69.25) mm, rotated rx -180 ry 0 rz -180 deg; joints [-27.726, 48.884, -77.477, 30.905, 115.065, 14.23]
  MoveL 4255 to (228.27, 35.88, 69.25) mm, rotated rx -180 ry 0 rz -180 deg; joints [-27.726, 48.884, -77.477, 30.905, 115.065, 14.23]
  Call Extruder(199.07188)
  MoveL 4256 to (228.52, 35.93, 69.25) mm, rotated rx -180 ry 0 rz 180 deg; joints [-27.673, 48.909, -77.477, 30.841, 115.056, 14.191]
  MoveL 4257 to (228.52, 35.93, 69.25) mm, rotated rx -180 ry 0 rz 180 deg; joints [-27.673, 48.909, -77.477, 30.841, 115.056, 14.191]
  Call Extruder(199.20947)
  MoveL 4258 to (228.77, 35.98, 69.25) mm, rotated rx 180 ry 0 rz 180 deg; joints [-27.62, 48.934, -77.477, 30.779, 115.047, 14.153]
  MoveL 4259 to (228.77, 35.98, 69.25) mm, rotated rx 180 ry 0 rz 180 deg; joints [-27.62, 48.934, -77.477, 30.779, 115.047, 14.153]
  Call Extruder(199.32318)
  MoveL 4260 to (228.97, 36.03, 69.25) mm, rotated rx -180 ry 0 rz 180 deg; joints [-27.579, 48.955, -77.477, 30.73, 115.039, 14.123]
  MoveL 4261 to (228.97, 36.03, 69.25) mm, rotated rx -180 ry 0 rz 180 deg; joints [-27.579, 48.955, -77.477, 30.73, 115.039, 14.123]
  Call Extruder(199.43735)
  MoveL 4262 to (229.18, 36.07, 69.25) mm, rotated rx -180 ry 0 rz -180 deg; joints [-27.539, 48.975, -77.477, 30.682, 115.031, 14.093]
  MoveL 4263 to (229.18, 36.07, 69.25) mm, rotated rx -180 ry 0 rz -180 deg; joints [-27.539, 48.975, -77.477, 30.682, 115.031, 14.093]
  Call Extruder(199.55198)
  MoveL 4264 to (229.38, 36.12, 69.25) mm, rotated rx 180 ry 0 rz 180 deg; joints [-27.499, 48.996, -77.476, 30.634, 115.023, 14.063]
  MoveL 4265 to (229.38, 36.12, 69.25) mm, rotated rx 180 ry 0 rz 180 deg; joints [-27.499, 48.996, -77.476, 30.634, 115.023, 14.063]
  Call Extruder(199.66705)
  MoveL 4266 to (229.59, 36.16, 69.25) mm, rotated rx 180 ry 0 rz 180 deg; joints [-27.458, 49.017, -77.476, 30.586, 115.015, 14.033]
  MoveL 4267 to (229.59, 36.16, 69.25) mm, rotated rx 180 ry 0 rz 180 deg; joints [-27.458, 49.017, -77.476, 30.586, 115.015, 14.033]
  Call Extruder(199.78928)
  MoveL 4268 to (229.8, 36.22, 69.25) mm, rotated rx -180 ry 0 rz 180 deg; joints [-27.423, 49.039, -77.476, 30.543, 115.004, 14.004]
  MoveL 4269 to (229.8, 36.22, 69.25) mm, rotated rx -180 ry 0 rz 180 deg; joints [-27.423, 49.039, -77.476, 30.543, 115.004, 14.004]
  Call Extruder(199.91895)
  MoveL 4270 to (230.02, 36.28, 69.25) mm, rotated rx -180 ry 0 rz 180 deg; joints [-27.392, 49.063, -77.475, 30.504, 114.991, 13.976]
  MoveL 4271 to (230.02, 36.28, 69.25) mm, rotated rx -180 ry 0 rz 180 deg; joints [-27.392, 49.063, -77.475, 30.504, 114.991, 13.976]
  Call Extruder(200.04918)
  MoveL 4272 to (230.25, 36.35, 69.25) mm, rotated rx -180 ry 0 rz 180 deg; joints [-27.361, 49.086, -77.475, 30.465, 114.977, 13.949]
  MoveL 4273 to (230.25, 36.35, 69.25) mm, rotated rx -180 ry 0 rz 180 deg; joints [-27.361, 49.086, -77.475, 30.465, 114.977, 13.949]
  Call Extruder(200.17998)
  MoveL 4274 to (230.47, 36.42, 69.25) mm, rotated rx 180 ry 0 rz 180 deg; joints [-27.33, 49.11, -77.475, 30.426, 114.964, 13.922]
  MoveL 4275 to (230.47, 36.42, 69.25) mm, rotated rx 180 ry 0 rz 180 deg; joints [-27.33, 49.11, -77.475, 30.426, 114.964, 13.922]
  Call Extruder(200.31134)
  MoveL 4276 to (230.69, 36.49, 69.25) mm, rotated rx -180 ry 0 rz 180 deg; joints [-27.299, 49.134, -77.474, 30.388, 114.951, 13.894]
  MoveL 4277 to (230.69, 36.49, 69.25) mm, rotated rx -180 ry 0 rz 180 deg; joints [-27.299, 49.134, -77.474, 30.388, 114.951, 13.894]
  Call Extruder(200.42676)
  MoveL 4278 to (230.89, 36.55, 69.25) mm, rotated rx 180 ry 0 rz 180 deg; joints [-27.275, 49.154, -77.474, 30.357, 114.938, 13.872]
  MoveL 4279 to (230.89, 36.55, 69.25) mm, rotated rx 180 ry 0 rz 180 deg; joints [-27.275, 49.154, -77.474, 30.357, 114.938, 13.872]
  Call Extruder(200.54265)
  MoveL 4280 to (231.08, 36.61, 69.25) mm, rotated rx -180 ry 0 rz 180 deg; joints [-27.252, 49.175, -77.474, 30.327, 114.926, 13.85]
  MoveL 4281 to (231.08, 36.61, 69.25) mm, rotated rx -180 ry 0 rz 180 deg; joints [-27.252, 49.175, -77.474, 30.327, 114.926, 13.85]
  Call Extruder(200.65547)
  MoveL 4282 to (231.27, 36.67, 69.25) mm, rotated rx -180 ry 0 rz 180 deg; joints [-27.229, 49.195, -77.473, 30.298, 114.914, 13.828]
  MoveL 4283 to (231.27, 36.67, 69.25) mm, rotated rx -180 ry 0 rz 180 deg; joints [-27.229, 49.195, -77.473, 30.298, 114.914, 13.828]
  Call Extruder(200.76517)
  MoveL 4284 to (231.46, 36.73, 69.25) mm, rotated rx -180 ry 0 rz 180 deg; joints [-27.207, 49.215, -77.473, 30.27, 114.902, 13.807]
  MoveL 4285 to (231.46, 36.73, 69.25) mm, rotated rx -180 ry 0 rz 180 deg; joints [-27.207, 49.215, -77.473, 30.27, 114.902, 13.807]
  Call Extruder(200.87528)
  MoveL 4286 to (231.64, 36.79, 69.25) mm, rotated rx -180 ry 0 rz 180 deg; joints [-27.185, 49.234, -77.472, 30.242, 114.89, 13.786]
  MoveL 4287 to (231.64, 36.79, 69.25) mm, rotated rx -180 ry 0 rz 180 deg; joints [-27.185, 49.234, -77.472, 30.242, 114.89, 13.786]
  Call Extruder(201.05724)
  MoveL 4288 to (231.93, 36.91, 69.25) mm, rotated rx -180 ry 0 rz -180 deg; joints [-27.167, 49.266, -77.472, 30.214, 114.866, 13.76]
  MoveL 4289 to (231.93, 36.91, 69.25) mm, rotated rx -180 ry 0 rz -180 deg; joints [-27.167, 49.266, -77.472, 30.214, 114.866, 13.76]
  Call Extruder(201.23996)
  MoveL 4290 to (232.22, 37.04, 69.25) mm, rotated rx 180 ry 0 rz 180 deg; joints [-27.149, 49.299, -77.471, 30.187, 114.842, 13.733]
  MoveL 4291 to (232.22, 37.04, 69.25) mm, rotated rx 180 ry 0 rz 180 deg; joints [-27.149, 49.299, -77.471, 30.187, 114.842, 13.733]
  Call Extruder(201.41037)
  MoveL 4292 to (232.49, 37.15, 69.25) mm, rotated rx 180 ry 0 rz -180 deg; joints [-27.133, 49.328, -77.47, 30.164, 114.819, 13.709]
  MoveL 4293 to (232.49, 37.15, 69.25) mm, rotated rx 180 ry 0 rz -180 deg; joints [-27.133, 49.328, -77.47, 30.164, 114.819, 13.709]
  Call Extruder(201.56837)
  MoveL 4294 to (232.74, 37.26, 69.25) mm, rotated rx 180 ry 0 rz 180 deg; joints [-27.121, 49.356, -77.47, 30.143, 114.797, 13.688]
  MoveL 4295 to (232.74, 37.26, 69.25) mm, rotated rx 180 ry 0 rz 180 deg; joints [-27.121, 49.356, -77.47, 30.143, 114.797, 13.688]
  Call Extruder(201.72697)
  MoveL 4296 to (232.99, 37.36, 69.25) mm, rotated rx -180 ry 0 rz 180 deg; joints [-27.108, 49.384, -77.469, 30.123, 114.776, 13.666]
  MoveL 4297 to (232.99, 37.36, 69.25) mm, rotated rx -180 ry 0 rz 180 deg; joints [-27.108, 49.384, -77.469, 30.123, 114.776, 13.666]
  Call Extruder(201.93314)
  MoveL 4298 to (233.29, 37.54, 69.25) mm, rotated rx -180 ry 0 rz 180 deg; joints [-27.12, 49.42, -77.468, 30.127, 114.741, 13.651]
  MoveL 4299 to (233.29, 37.54, 69.25) mm, rotated rx -180 ry 0 rz 180 deg; joints [-27.12, 49.42, -77.468, 30.127, 114.741, 13.651]
  Call Extruder(202.14008)
  MoveL 4300 to (233.6, 37.71, 69.25) mm, rotated rx -180 ry 0 rz -180 deg; joints [-27.132, 49.455, -77.467, 30.132, 114.706, 13.637]
  MoveL 4301 to (233.6, 37.71, 69.25) mm, rotated rx -180 ry 0 rz -180 deg; joints [-27.132, 49.455, -77.467, 30.132, 114.706, 13.637]
  Call Extruder(202.34781)
  MoveL 4302 to (233.9, 37.89, 69.25) mm, rotated rx -180 ry 0 rz 180 deg; joints [-27.144, 49.491, -77.466, 30.136, 114.672, 13.622]
  MoveL 4303 to (233.9, 37.89, 69.25) mm, rotated rx -180 ry 0 rz 180 deg; joints [-27.144, 49.491, -77.466, 30.136, 114.672, 13.622]
  Call Extruder(202.55631)
  MoveL 4304 to (234.21, 38.07, 69.25) mm, rotated rx 180 ry 0 rz -180 deg; joints [-27.156, 49.527, -77.465, 30.141, 114.637, 13.607]
  MoveL 4305 to (234.21, 38.07, 69.25) mm, rotated rx 180 ry 0 rz -180 deg; joints [-27.156, 49.527, -77.465, 30.141, 114.637, 13.607]
  Call Extruder(202.73585)
  MoveL 4306 to (234.45, 38.24, 69.25) mm, rotated rx -180 ry 0 rz 180 deg; joints [-27.187, 49.557, -77.464, 30.166, 114.603, 13.603]
  MoveL 4307 to (234.45, 38.24, 69.25) mm, rotated rx -180 ry 0 rz 180 deg; joints [-27.187, 49.557, -77.464, 30.166, 114.603, 13.603]
  Call Extruder(203.06927)
  MoveL 4308 to (234.9, 38.57, 69.25) mm, rotated rx -180 ry 0 rz 180 deg; joints [-27.245, 49.613, -77.462, 30.215, 114.539, 13.597]
  MoveL 4309 to (234.9, 38.57, 69.25) mm, rotated rx -180 ry 0 rz 180 deg; joints [-27.245, 49.613, -77.462, 30.215, 114.539, 13.597]
  Call Extruder(203.40387)
  MoveL 4310 to (235.35, 38.9, 69.25) mm, rotated rx 180 ry 0 rz 180 deg; joints [-27.302, 49.669, -77.46, 30.263, 114.475, 13.59]
  Call Extruder(204.23182)
  MoveL 4311 to (236.39, 39.81, 69.25) mm, rotated rx -180 ry 0 rz 180 deg; joints [-27.525, 49.805, -77.455, 30.468, 114.301, 13.61]
  Call Extruder(205.05976)
  MoveL 4312 to (237.3, 40.85, 69.25) mm, rotated rx -180 ry 0 rz 180 deg; joints [-27.851, 49.936, -77.449, 30.785, 114.107, 13.676]
  Call Extruder(205.22706)
  MoveL 4313 to (237.47, 41.07, 69.25) mm, rotated rx 180 ry 0 rz -180 deg; joints [-27.932, 49.961, -77.448, 30.865, 114.065, 13.696]
  MoveL 4314 to (237.47, 41.07, 69.25) mm, rotated rx 180 ry 0 rz -180 deg; joints [-27.932, 49.961, -77.448, 30.865, 114.065, 13.696]
  Call Extruder(205.56048)
  MoveL 4315 to (237.79, 41.52, 69.25) mm, rotated rx -180 ry 0 rz 180 deg; joints [-28.091, 50.012, -77.445, 31.022, 113.982, 13.735]
  MoveL 4316 to (237.79, 41.52, 69.25) mm, rotated rx -180 ry 0 rz 180 deg; joints [-28.091, 50.012, -77.445, 31.022, 113.982, 13.735]
  Call Extruder(205.89270)
  MoveL 4317 to (238.12, 41.98, 69.25) mm, rotated rx -180 ry 0 rz -180 deg; joints [-28.249, 50.062, -77.443, 31.177, 113.899, 13.773]
  MoveL 4318 to (238.12, 41.98, 69.25) mm, rotated rx -180 ry 0 rz -180 deg; joints [-28.249, 50.062, -77.443, 31.177, 113.899, 13.773]
  Call Extruder(206.01040)
  MoveL 4319 to (238.22, 42.15, 69.25) mm, rotated rx 180 ry 0 rz 180 deg; joints [-28.315, 50.079, -77.442, 31.244, 113.868, 13.792]
  MoveL 4320 to (238.22, 42.15, 69.25) mm, rotated rx 180 ry 0 rz 180 deg; joints [-28.315, 50.079, -77.442, 31.244, 113.868, 13.792]
  Call Extruder(206.21813)
  MoveL 4321 to (238.4, 42.45, 69.25) mm, rotated rx -180 ry 0 rz 180 deg; joints [-28.434, 50.109, -77.44, 31.362, 113.812, 13.825]
  MoveL 4322 to (238.4, 42.45, 69.25) mm, rotated rx -180 ry 0 rz 180 deg; joints [-28.434, 50.109, -77.44, 31.362, 113.812, 13.825]
  Call Extruder(206.42507)
  MoveL 4323 to (238.57, 42.75, 69.25) mm, rotated rx 180 ry 0 rz 180 deg; joints [-28.552, 50.14, -77.439, 31.48, 113.757, 13.857]
  MoveL 4324 to (238.57, 42.75, 69.25) mm, rotated rx 180 ry 0 rz 180 deg; joints [-28.552, 50.14, -77.439, 31.48, 113.757, 13.857]
  Call Extruder(206.63124)
  MoveL 4325 to (238.75, 43.06, 69.25) mm, rotated rx 180 ry 0 rz 180 deg; joints [-28.669, 50.17, -77.437, 31.597, 113.702, 13.889]
  MoveL 4326 to (238.75, 43.06, 69.25) mm, rotated rx 180 ry 0 rz 180 deg; joints [-28.669, 50.17, -77.437, 31.597, 113.702, 13.889]
  Call Extruder(206.81293)
  MoveL 4327 to (238.89, 43.33, 69.25) mm, rotated rx -180 ry 0 rz 180 deg; joints [-28.78, 50.196, -77.436, 31.709, 113.652, 13.921]
  MoveL 4328 to (238.89, 43.33, 69.25) mm, rotated rx -180 ry 0 rz 180 deg; joints [-28.78, 50.196, -77.436, 31.709, 113.652, 13.921]
  Call Extruder(206.97094)
  MoveL 4329 to (239, 43.58, 69.25) mm, rotated rx 180 ry 0 rz 180 deg; joints [-28.886, 50.217, -77.434, 31.816, 113.607, 13.953]
  MoveL 4330 to (239, 43.58, 69.25) mm, rotated rx 180 ry 0 rz 180 deg; joints [-28.886, 50.217, -77.434, 31.816, 113.607, 13.953]
  Call Extruder(207.12835)
  MoveL 4331 to (239.11, 43.83, 69.25) mm, rotated rx -180 ry 0 rz 180 deg; joints [-28.991, 50.238, -77.433, 31.922, 113.562, 13.984]
  MoveL 4332 to (239.11, 43.83, 69.25) mm, rotated rx -180 ry 0 rz 180 deg; joints [-28.991, 50.238, -77.433, 31.922, 113.562, 13.984]
  Call Extruder(207.31106)
  MoveL 4333 to (239.23, 44.13, 69.25) mm, rotated rx -180 ry 0 rz -180 deg; joints [-29.116, 50.263, -77.432, 32.048, 113.51, 14.022]
  MoveL 4334 to (239.23, 44.13, 69.25) mm, rotated rx -180 ry 0 rz -180 deg; joints [-29.116, 50.263, -77.432, 32.048, 113.51, 14.022]
  Call Extruder(207.49302)
  MoveL 4335 to (239.35, 44.42, 69.25) mm, rotated rx -180 ry 0 rz 180 deg; joints [-29.24, 50.288, -77.43, 32.172, 113.458, 14.059]
  MoveL 4336 to (239.35, 44.42, 69.25) mm, rotated rx -180 ry 0 rz 180 deg; joints [-29.24, 50.288, -77.43, 32.172, 113.458, 14.059]
  Call Extruder(207.64035)
  MoveL 4337 to (239.44, 44.66, 69.25) mm, rotated rx -180 ry 0 rz 180 deg; joints [-29.343, 50.308, -77.429, 32.277, 113.415, 14.09]
  MoveL 4338 to (239.44, 44.66, 69.25) mm, rotated rx -180 ry 0 rz 180 deg; joints [-29.343, 50.308, -77.429, 32.277, 113.415, 14.09]
  Call Extruder(207.75359)
  MoveL 4339 to (239.5, 44.85, 69.25) mm, rotated rx -180 ry 0 rz 180 deg; joints [-29.428, 50.322, -77.428, 32.363, 113.381, 14.116]
  MoveL 4340 to (239.5, 44.85, 69.25) mm, rotated rx -180 ry 0 rz 180 deg; joints [-29.428, 50.322, -77.428, 32.363, 113.381, 14.116]
  Call Extruder(207.86638)
  MoveL 4341 to (239.56, 45.03, 69.25) mm, rotated rx -180 ry 0 rz 180 deg; joints [-29.512, 50.337, -77.427, 32.448, 113.348, 14.142]
  MoveL 4342 to (239.56, 45.03, 69.25) mm, rotated rx -180 ry 0 rz 180 deg; joints [-29.512, 50.337, -77.427, 32.448, 113.348, 14.142]
  Call Extruder(207.97872)
  MoveL 4343 to (239.62, 45.22, 69.25) mm, rotated rx 180 ry 0 rz 180 deg; joints [-29.596, 50.352, -77.426, 32.533, 113.314, 14.168]
  MoveL 4344 to (239.62, 45.22, 69.25) mm, rotated rx 180 ry 0 rz 180 deg; joints [-29.596, 50.352, -77.426, 32.533, 113.314, 14.168]
  Call Extruder(208.09063)
  MoveL 4345 to (239.68, 45.41, 69.25) mm, rotated rx 180 ry 0 rz 180 deg; joints [-29.679, 50.366, -77.425, 32.617, 113.28, 14.194]
  MoveL 4346 to (239.68, 45.41, 69.25) mm, rotated rx 180 ry 0 rz 180 deg; joints [-29.679, 50.366, -77.425, 32.617, 113.28, 14.194]
  Call Extruder(208.21203)
  MoveL 4347 to (239.75, 45.62, 69.25) mm, rotated rx -180 ry 0 rz 180 deg; joints [-29.77, 50.382, -77.424, 32.71, 113.244, 14.222]
  MoveL 4348 to (239.75, 45.62, 69.25) mm, rotated rx -180 ry 0 rz 180 deg; joints [-29.77, 50.382, -77.424, 32.71, 113.244, 14.222]
  Call Extruder(208.34282)
  MoveL 4349 to (239.82, 45.84, 69.25) mm, rotated rx -180 ry 0 rz 180 deg; joints [-29.871, 50.399, -77.423, 32.811, 113.204, 14.253]
  MoveL 4350 to (239.82, 45.84, 69.25) mm, rotated rx -180 ry 0 rz 180 deg; joints [-29.871, 50.399, -77.423, 32.811, 113.204, 14.253]
  Call Extruder(208.47304)
  MoveL 4351 to (239.88, 46.06, 69.25) mm, rotated rx -180 ry 0 rz 180 deg; joints [-29.97, 50.416, -77.422, 32.912, 113.164, 14.284]
  MoveL 4352 to (239.88, 46.06, 69.25) mm, rotated rx -180 ry 0 rz 180 deg; joints [-29.97, 50.416, -77.422, 32.912, 113.164, 14.284]
  Call Extruder(208.60270)
  MoveL 4353 to (239.95, 46.29, 69.25) mm, rotated rx -180 ry 0 rz 180 deg; joints [-30.069, 50.433, -77.421, 33.012, 113.124, 14.314]
  MoveL 4354 to (239.95, 46.29, 69.25) mm, rotated rx -180 ry 0 rz 180 deg; joints [-30.069, 50.433, -77.421, 33.012, 113.124, 14.314]
  Call Extruder(208.73180)
  MoveL 4355 to (240.02, 46.51, 69.25) mm, rotated rx 180 ry 0 rz 180 deg; joints [-30.168, 50.45, -77.42, 33.113, 113.085, 14.345]
  MoveL 4356 to (240.02, 46.51, 69.25) mm, rotated rx 180 ry 0 rz 180 deg; joints [-30.168, 50.45, -77.42, 33.113, 113.085, 14.345]
  Call Extruder(208.84685)
  MoveL 4357 to (240.06, 46.72, 69.25) mm, rotated rx -180 ry 0 rz 180 deg; joints [-30.263, 50.464, -77.419, 33.209, 113.049, 14.375]
  MoveL 4358 to (240.06, 46.72, 69.25) mm, rotated rx -180 ry 0 rz 180 deg; joints [-30.263, 50.464, -77.419, 33.209, 113.049, 14.375]
  Call Extruder(208.96145)
  MoveL 4359 to (240.11, 46.92, 69.25) mm, rotated rx 180 ry 0 rz 180 deg; joints [-30.358, 50.478, -77.418, 33.305, 113.012, 14.405]
  MoveL 4360 to (240.11, 46.92, 69.25) mm, rotated rx 180 ry 0 rz 180 deg; joints [-30.358, 50.478, -77.418, 33.305, 113.012, 14.405]
  Call Extruder(209.07560)
  MoveL 4361 to (240.15, 47.12, 69.25) mm, rotated rx 180 ry 0 rz 180 deg; joints [-30.453, 50.493, -77.417, 33.402, 112.976, 14.435]
  MoveL 4362 to (240.15, 47.12, 69.25) mm, rotated rx 180 ry 0 rz 180 deg; joints [-30.453, 50.493, -77.417, 33.402, 112.976, 14.435]
  Call Extruder(209.18930)
  MoveL 4363 to (240.2, 47.33, 69.25) mm, rotated rx 180 ry 0 rz -180 deg; joints [-30.548, 50.507, -77.416, 33.498, 112.94, 14.465]
  MoveL 4364 to (240.2, 47.33, 69.25) mm, rotated rx 180 ry 0 rz -180 deg; joints [-30.548, 50.507, -77.416, 33.498, 112.94, 14.465]
  Call Extruder(209.31471)
  MoveL 4365 to (240.24, 47.55, 69.25) mm, rotated rx -180 ry 0 rz 180 deg; joints [-30.653, 50.522, -77.415, 33.604, 112.9, 14.497]
  MoveL 4366 to (240.24, 47.55, 69.25) mm, rotated rx -180 ry 0 rz 180 deg; joints [-30.653, 50.522, -77.415, 33.604, 112.9, 14.497]
  Call Extruder(209.45169)
  MoveL 4367 to (240.29, 47.8, 69.25) mm, rotated rx -180 ry 0 rz 180 deg; joints [-30.768, 50.539, -77.414, 33.721, 112.856, 14.534]
  MoveL 4368 to (240.29, 47.8, 69.25) mm, rotated rx -180 ry 0 rz 180 deg; joints [-30.768, 50.539, -77.414, 33.721, 112.856, 14.534]
  Call Extruder(209.58805)
  MoveL 4369 to (240.34, 48.05, 69.25) mm, rotated rx -180 ry 0 rz 180 deg; joints [-30.884, 50.556, -77.413, 33.839, 112.812, 14.57]
  MoveL 4370 to (240.34, 48.05, 69.25) mm, rotated rx -180 ry 0 rz 180 deg; joints [-30.884, 50.556, -77.413, 33.839, 112.812, 14.57]
  Call Extruder(209.72381)
  MoveL 4371 to (240.39, 48.3, 69.25) mm, rotated rx 180 ry 0 rz -180 deg; joints [-30.999, 50.573, -77.411, 33.955, 112.767, 14.606]
  MoveL 4372 to (240.39, 48.3, 69.25) mm, rotated rx 180 ry 0 rz -180 deg; joints [-30.999, 50.573, -77.411, 33.955, 112.767, 14.606]
  Call Extruder(209.85896)
  MoveL 4373 to (240.44, 48.55, 69.25) mm, rotated rx -180 ry 0 rz 180 deg; joints [-31.114, 50.59, -77.41, 34.072, 112.723, 14.641]
  MoveL 4374 to (240.44, 48.55, 69.25) mm, rotated rx -180 ry 0 rz 180 deg; joints [-31.114, 50.59, -77.41, 34.072, 112.723, 14.641]
  Call Extruder(209.99349)
  MoveL 4375 to (240.49, 48.8, 69.25) mm, rotated rx -180 ry 0 rz 180 deg; joints [-31.228, 50.607, -77.409, 34.187, 112.679, 14.676]
  MoveL 4376 to (240.49, 48.8, 69.25) mm, rotated rx -180 ry 0 rz 180 deg; joints [-31.228, 50.607, -77.409, 34.187, 112.679, 14.676]
  Call Extruder(210.12742)
  MoveL 4377 to (240.54, 49.05, 69.25) mm, rotated rx -180 ry 0 rz 180 deg; joints [-31.342, 50.624, -77.408, 34.302, 112.635, 14.711]
  MoveL 4378 to (240.54, 49.05, 69.25) mm, rotated rx -180 ry 0 rz 180 deg; joints [-31.342, 50.624, -77.408, 34.302, 112.635, 14.711]
  Call Extruder(210.27529)
  MoveL 4379 to (240.59, 49.33, 69.25) mm, rotated rx 180 ry 0 rz 180 deg; joints [-31.47, 50.643, -77.406, 34.431, 112.586, 14.751]
  MoveL 4380 to (240.59, 49.33, 69.25) mm, rotated rx 180 ry 0 rz 180 deg; joints [-31.47, 50.643, -77.406, 34.431, 112.586, 14.751]
  Call Extruder(210.43703)
  MoveL 4381 to (240.64, 49.63, 69.25) mm, rotated rx -180 ry 0 rz 180 deg; joints [-31.612, 50.663, -77.405, 34.575, 112.532, 14.795]
  MoveL 4382 to (240.64, 49.63, 69.25) mm, rotated rx -180 ry 0 rz 180 deg; joints [-31.612, 50.663, -77.405, 34.575, 112.532, 14.795]
  Call Extruder(210.59805)
  MoveL 4383 to (240.69, 49.94, 69.25) mm, rotated rx -180 ry 0 rz -180 deg; joints [-31.755, 50.683, -77.403, 34.719, 112.478, 14.838]
  MoveL 4384 to (240.69, 49.94, 69.25) mm, rotated rx -180 ry 0 rz -180 deg; joints [-31.755, 50.683, -77.403, 34.719, 112.478, 14.838]
  Call Extruder(210.75834)
  MoveL 4385 to (240.74, 50.24, 69.25) mm, rotated rx -180 ry 0 rz 180 deg; joints [-31.895, 50.703, -77.402, 34.861, 112.424, 14.881]
  MoveL 4386 to (240.74, 50.24, 69.25) mm, rotated rx -180 ry 0 rz 180 deg; joints [-31.895, 50.703, -77.402, 34.861, 112.424, 14.881]
  Call Extruder(210.91790)
  MoveL 4387 to (240.78, 50.55, 69.25) mm, rotated rx -180 ry 0 rz 180 deg; joints [-32.036, 50.723, -77.4, 35.003, 112.37, 14.924]
  MoveL 4388 to (240.78, 50.55, 69.25) mm, rotated rx -180 ry 0 rz 180 deg; joints [-32.036, 50.723, -77.4, 35.003, 112.37, 14.924]
  Call Extruder(211.07673)
  MoveL 4389 to (240.83, 50.86, 69.25) mm, rotated rx -180 ry 0 rz 180 deg; joints [-32.176, 50.743, -77.399, 35.145, 112.316, 14.966]
  MoveL 4390 to (240.83, 50.86, 69.25) mm, rotated rx -180 ry 0 rz 180 deg; joints [-32.176, 50.743, -77.399, 35.145, 112.316, 14.966]
  Call Extruder(211.25540)
  MoveL 4391 to (240.88, 51.2, 69.25) mm, rotated rx -180 ry 0 rz 180 deg; joints [-32.337, 50.766, -77.397, 35.306, 112.255, 15.015]
  MoveL 4392 to (240.88, 51.2, 69.25) mm, rotated rx -180 ry 0 rz 180 deg; joints [-32.337, 50.766, -77.397, 35.306, 112.255, 15.015]
  Call Extruder(211.45384)
  MoveL 4393 to (240.93, 51.59, 69.25) mm, rotated rx -180 ry 0 rz 180 deg; joints [-32.518, 50.79, -77.395, 35.489, 112.187, 15.069]
  MoveL 4394 to (240.93, 51.59, 69.25) mm, rotated rx -180 ry 0 rz 180 deg; joints [-32.518, 50.79, -77.395, 35.489, 112.187, 15.069]
  Call Extruder(211.65142)
  MoveL 4395 to (240.97, 51.98, 69.25) mm, rotated rx -180 ry 0 rz 180 deg; joints [-32.697, 50.815, -77.393, 35.67, 112.118, 15.123]
  MoveL 4396 to (240.97, 51.98, 69.25) mm, rotated rx -180 ry 0 rz 180 deg; joints [-32.697, 50.815, -77.393, 35.67, 112.118, 15.123]
  Call Extruder(211.84813)
  MoveL 4397 to (241.02, 52.36, 69.25) mm, rotated rx 180 ry 0 rz 180 deg; joints [-32.876, 50.839, -77.391, 35.85, 112.05, 15.177]
  MoveL 4398 to (241.02, 52.36, 69.25) mm, rotated rx 180 ry 0 rz 180 deg; joints [-32.876, 50.839, -77.391, 35.85, 112.05, 15.177]
  Call Extruder(212.04396)
  MoveL 4399 to (241.06, 52.75, 69.25) mm, rotated rx 180 ry 0 rz 180 deg; joints [-33.055, 50.864, -77.389, 36.029, 111.982, 15.229]
  MoveL 4400 to (241.06, 52.75, 69.25) mm, rotated rx 180 ry 0 rz 180 deg; joints [-33.055, 50.864, -77.389, 36.029, 111.982, 15.229]
  Call Extruder(212.33940)
  MoveL 4401 to (241.11, 53.34, 69.25) mm, rotated rx 180 ry 0 rz 180 deg; joints [-33.331, 50.9, -77.386, 36.308, 111.878, 15.312]
  MoveL 4402 to (241.11, 53.34, 69.25) mm, rotated rx 180 ry 0 rz 180 deg; joints [-33.331, 50.9, -77.386, 36.308, 111.878, 15.312]
  Call Extruder(212.63351)
  MoveL 4403 to (241.15, 53.93, 69.25) mm, rotated rx -180 ry 0 rz 180 deg; joints [-33.606, 50.935, -77.383, 36.584, 111.774, 15.393]
  MoveL 4404 to (241.15, 53.93, 69.25) mm, rotated rx -180 ry 0 rz 180 deg; joints [-33.606, 50.935, -77.383, 36.584, 111.774, 15.393]
  Call Extruder(212.92629)
  MoveL 4405 to (241.2, 54.52, 69.25) mm, rotated rx 180 ry 0 rz -180 deg; joints [-33.878, 50.972, -77.38, 36.857, 111.67, 15.473]
  MoveL 4406 to (241.2, 54.52, 69.25) mm, rotated rx 180 ry 0 rz -180 deg; joints [-33.878, 50.972, -77.38, 36.857, 111.67, 15.473]
  Call Extruder(213.49974)
  MoveL 4407 to (241.25, 55.68, 69.25) mm, rotated rx -180 ry 0 rz 180 deg; joints [-34.425, 51.04, -77.374, 37.405, 111.464, 15.633]
  MoveL 4408 to (241.25, 55.68, 69.25) mm, rotated rx -180 ry 0 rz 180 deg; joints [-34.425, 51.04, -77.374, 37.405, 111.464, 15.633]
  Call Extruder(214.21357)
  MoveL 4409 to (241.29, 57.14, 69.25) mm, rotated rx 180 ry 0 rz 180 deg; joints [-35.104, 51.125, -77.366, 38.085, 111.207, 15.827]
  Call Extruder(256.27845)
  MoveL 4410 to (241.29, 142.86, 69.25) mm, rotated rx -180 ry 0 rz 180 deg; joints [-60.361, 57, -75.967, 61.715, 99.25, 16.631]
  Call Extruder(256.70688)
  MoveL 4411 to (241.27, 143.74, 69.25) mm, rotated rx 180 ry 0 rz -180 deg; joints [-60.516, 57.062, -75.942, 61.853, 99.164, 16.578]
  MoveL 4412 to (241.27, 143.74, 69.25) mm, rotated rx 180 ry 0 rz -180 deg; joints [-60.516, 57.062, -75.942, 61.853, 99.164, 16.578]
  Call Extruder(257.28033)
  MoveL 4413 to (241.22, 144.9, 69.25) mm, rotated rx -180 ry 0 rz 180 deg; joints [-60.726, 57.143, -75.908, 62.042, 99.05, 16.507]
  MoveL 4414 to (241.22, 144.9, 69.25) mm, rotated rx -180 ry 0 rz 180 deg; joints [-60.726, 57.143, -75.908, 62.042, 99.05, 16.507]
  Call Extruder(257.71467)
  MoveL 4415 to (241.18, 145.77, 69.25) mm, rotated rx 180 ry 0 rz 180 deg; joints [-60.887, 57.203, -75.882, 62.186, 98.964, 16.455]
  MoveL 4416 to (241.18, 145.77, 69.25) mm, rotated rx 180 ry 0 rz 180 deg; joints [-60.887, 57.203, -75.882, 62.186, 98.964, 16.455]
  Call Extruder(258.00878)
  MoveL 4417 to (241.13, 146.36, 69.25) mm, rotated rx 180 ry 0 rz -180 deg; joints [-61, 57.243, -75.865, 62.287, 98.906, 16.421]
  MoveL 4418 to (241.13, 146.36, 69.25) mm, rotated rx 180 ry 0 rz -180 deg; joints [-61, 57.243, -75.865, 62.287, 98.906, 16.421]
  Call Extruder(258.30422)
  MoveL 4419 to (241.09, 146.95, 69.25) mm, rotated rx 180 ry 0 rz 180 deg; joints [-61.111, 57.283, -75.847, 62.387, 98.848, 16.386]
  MoveL 4420 to (241.09, 146.95, 69.25) mm, rotated rx 180 ry 0 rz 180 deg; joints [-61.111, 57.283, -75.847, 62.387, 98.848, 16.386]
  Call Extruder(258.55047)
  MoveL 4421 to (241.04, 147.44, 69.25) mm, rotated rx -180 ry 0 rz -180 deg; joints [-61.205, 57.316, -75.833, 62.472, 98.799, 16.357]
  MoveL 4422 to (241.04, 147.44, 69.25) mm, rotated rx -180 ry 0 rz -180 deg; joints [-61.205, 57.316, -75.833, 62.472, 98.799, 16.357]
  Call Extruder(258.74718)
  MoveL 4423 to (240.99, 147.83, 69.25) mm, rotated rx 180 ry 0 rz -180 deg; joints [-61.282, 57.342, -75.822, 62.542, 98.76, 16.336]
  MoveL 4424 to (240.99, 147.83, 69.25) mm, rotated rx 180 ry 0 rz -180 deg; joints [-61.282, 57.342, -75.822, 62.542, 98.76, 16.336]
  Call Extruder(258.94475)
  MoveL 4425 to (240.95, 148.22, 69.25) mm, rotated rx 180 ry 0 rz -180 deg; joints [-61.359, 57.368, -75.811, 62.611, 98.722, 16.314]
  MoveL 4426 to (240.95, 148.22, 69.25) mm, rotated rx 180 ry 0 rz -180 deg; joints [-61.359, 57.368, -75.811, 62.611, 98.722, 16.314]
  Call Extruder(259.14319)
  MoveL 4427 to (240.9, 148.6, 69.25) mm, rotated rx -180 ry 0 rz 180 deg; joints [-61.436, 57.393, -75.799, 62.681, 98.683, 16.292]
  MoveL 4428 to (240.9, 148.6, 69.25) mm, rotated rx -180 ry 0 rz 180 deg; joints [-61.436, 57.393, -75.799, 62.681, 98.683, 16.292]
  Call Extruder(259.34250)
  MoveL 4429 to (240.86, 148.99, 69.25) mm, rotated rx 180 ry 0 rz 180 deg; joints [-61.512, 57.419, -75.788, 62.75, 98.645, 16.27]
  MoveL 4430 to (240.86, 148.99, 69.25) mm, rotated rx 180 ry 0 rz 180 deg; joints [-61.512, 57.419, -75.788, 62.75, 98.645, 16.27]
  Call Extruder(259.50134)
  MoveL 4431 to (240.81, 149.3, 69.25) mm, rotated rx -180 ry 0 rz 180 deg; joints [-61.575, 57.439, -75.779, 62.808, 98.614, 16.253]
  MoveL 4432 to (240.81, 149.3, 69.25) mm, rotated rx -180 ry 0 rz 180 deg; joints [-61.575, 57.439, -75.779, 62.808, 98.614, 16.253]
  Call Extruder(259.66090)
  MoveL 4433 to (240.76, 149.6, 69.25) mm, rotated rx 180 ry 0 rz 180 deg; joints [-61.639, 57.459, -75.77, 62.865, 98.583, 16.237]
  MoveL 4434 to (240.76, 149.6, 69.25) mm, rotated rx 180 ry 0 rz 180 deg; joints [-61.639, 57.459, -75.77, 62.865, 98.583, 16.237]
  Call Extruder(259.82119)
  MoveL 4435 to (240.71, 149.91, 69.25) mm, rotated rx 180 ry 0 rz 180 deg; joints [-61.702, 57.478, -75.761, 62.923, 98.553, 16.22]
  MoveL 4436 to (240.71, 149.91, 69.25) mm, rotated rx 180 ry 0 rz 180 deg; joints [-61.702, 57.478, -75.761, 62.923, 98.553, 16.22]
  Call Extruder(259.98220)
  MoveL 4437 to (240.66, 150.21, 69.25) mm, rotated rx -180 ry 0 rz 180 deg; joints [-61.765, 57.498, -75.753, 62.98, 98.522, 16.203]
  MoveL 4438 to (240.66, 150.21, 69.25) mm, rotated rx -180 ry 0 rz 180 deg; joints [-61.765, 57.498, -75.753, 62.98, 98.522, 16.203]
  Call Extruder(260.14395)
  MoveL 4439 to (240.61, 150.52, 69.25) mm, rotated rx -180 ry 0 rz 180 deg; joints [-61.828, 57.518, -75.744, 63.037, 98.491, 16.186]
  MoveL 4440 to (240.61, 150.52, 69.25) mm, rotated rx -180 ry 0 rz 180 deg; joints [-61.828, 57.518, -75.744, 63.037, 98.491, 16.186]
  Call Extruder(260.30642)
  MoveL 4441 to (240.57, 150.83, 69.25) mm, rotated rx 180 ry 0 rz 180 deg; joints [-61.891, 57.538, -75.735, 63.095, 98.461, 16.169]
  MoveL 4442 to (240.57, 150.83, 69.25) mm, rotated rx 180 ry 0 rz 180 deg; joints [-61.891, 57.538, -75.735, 63.095, 98.461, 16.169]
  Call Extruder(260.44035)
  MoveL 4443 to (240.52, 151.07, 69.25) mm, rotated rx 180 ry 0 rz -180 deg; joints [-61.944, 57.554, -75.728, 63.144, 98.435, 16.156]
  MoveL 4444 to (240.52, 151.07, 69.25) mm, rotated rx 180 ry 0 rz -180 deg; joints [-61.944, 57.554, -75.728, 63.144, 98.435, 16.156]
  Call Extruder(260.57488)
  MoveL 4445 to (240.47, 151.32, 69.25) mm, rotated rx 180 ry 0 rz 180 deg; joints [-61.998, 57.569, -75.72, 63.193, 98.41, 16.143]
  MoveL 4446 to (240.47, 151.32, 69.25) mm, rotated rx 180 ry 0 rz 180 deg; joints [-61.998, 57.569, -75.72, 63.193, 98.41, 16.143]
  Call Extruder(260.71003)
  MoveL 4447 to (240.42, 151.57, 69.25) mm, rotated rx 180 ry 0 rz 180 deg; joints [-62.052, 57.585, -75.713, 63.242, 98.385, 16.13]
  MoveL 4448 to (240.42, 151.57, 69.25) mm, rotated rx 180 ry 0 rz 180 deg; joints [-62.052, 57.585, -75.713, 63.242, 98.385, 16.13]
  Call Extruder(260.84579)
  MoveL 4449 to (240.37, 151.82, 69.25) mm, rotated rx -180 ry 0 rz 180 deg; joints [-62.105, 57.601, -75.706, 63.291, 98.36, 16.117]
  MoveL 4450 to (240.37, 151.82, 69.25) mm, rotated rx -180 ry 0 rz 180 deg; joints [-62.105, 57.601, -75.706, 63.291, 98.36, 16.117]
  Call Extruder(260.98215)
  MoveL 4451 to (240.32, 152.07, 69.25) mm, rotated rx -180 ry 0 rz 180 deg; joints [-62.159, 57.617, -75.699, 63.34, 98.335, 16.104]
  MoveL 4452 to (240.32, 152.07, 69.25) mm, rotated rx -180 ry 0 rz 180 deg; joints [-62.159, 57.617, -75.699, 63.34, 98.335, 16.104]
  Call Extruder(261.11913)
  MoveL 4453 to (240.27, 152.32, 69.25) mm, rotated rx 180 ry 0 rz 180 deg; joints [-62.212, 57.632, -75.692, 63.389, 98.31, 16.091]
  MoveL 4454 to (240.27, 152.32, 69.25) mm, rotated rx 180 ry 0 rz 180 deg; joints [-62.212, 57.632, -75.692, 63.389, 98.31, 16.091]
  Call Extruder(261.25672)
  MoveL 4455 to (240.22, 152.57, 69.25) mm, rotated rx 180 ry 0 rz 180 deg; joints [-62.265, 57.648, -75.684, 63.437, 98.284, 16.077]
  MoveL 4456 to (240.22, 152.57, 69.25) mm, rotated rx 180 ry 0 rz 180 deg; joints [-62.265, 57.648, -75.684, 63.437, 98.284, 16.077]
  Call Extruder(261.37042)
  MoveL 4457 to (240.17, 152.77, 69.25) mm, rotated rx -180 ry 0 rz 180 deg; joints [-62.31, 57.661, -75.678, 63.478, 98.264, 16.067]
  MoveL 4458 to (240.17, 152.77, 69.25) mm, rotated rx -180 ry 0 rz 180 deg; joints [-62.31, 57.661, -75.678, 63.478, 98.264, 16.067]
  Call Extruder(261.48457)
  MoveL 4459 to (240.13, 152.98, 69.25) mm, rotated rx 180 ry 0 rz 180 deg; joints [-62.355, 57.674, -75.672, 63.519, 98.243, 16.056]
  MoveL 4460 to (240.13, 152.98, 69.25) mm, rotated rx 180 ry 0 rz 180 deg; joints [-62.355, 57.674, -75.672, 63.519, 98.243, 16.056]
  Call Extruder(261.59917)
  MoveL 4461 to (240.08, 153.18, 69.25) mm, rotated rx 180 ry 0 rz 180 deg; joints [-62.399, 57.687, -75.667, 63.56, 98.222, 16.045]
  MoveL 4462 to (240.08, 153.18, 69.25) mm, rotated rx 180 ry 0 rz 180 deg; joints [-62.399, 57.687, -75.667, 63.56, 98.222, 16.045]
  Call Extruder(261.71422)
  MoveL 4463 to (240.04, 153.39, 69.25) mm, rotated rx 180 ry 0 rz 180 deg; joints [-62.444, 57.699, -75.661, 63.601, 98.202, 16.034]
  MoveL 4464 to (240.04, 153.39, 69.25) mm, rotated rx 180 ry 0 rz 180 deg; joints [-62.444, 57.699, -75.661, 63.601, 98.202, 16.034]
  Call Extruder(261.83645)
  MoveL 4465 to (239.98, 153.6, 69.25) mm, rotated rx 180 ry 0 rz 180 deg; joints [-62.493, 57.712, -75.654, 63.646, 98.18, 16.024]
  MoveL 4466 to (239.98, 153.6, 69.25) mm, rotated rx 180 ry 0 rz 180 deg; joints [-62.493, 57.712, -75.654, 63.646, 98.18, 16.024]
  Call Extruder(261.96611)
  MoveL 4467 to (239.92, 153.82, 69.25) mm, rotated rx 180 ry 0 rz 180 deg; joints [-62.547, 57.726, -75.648, 63.696, 98.156, 16.014]
  MoveL 4468 to (239.92, 153.82, 69.25) mm, rotated rx 180 ry 0 rz 180 deg; joints [-62.547, 57.726, -75.648, 63.696, 98.156, 16.014]
  Call Extruder(262.09633)
  MoveL 4469 to (239.85, 154.05, 69.25) mm, rotated rx -180 ry 0 rz 180 deg; joints [-62.601, 57.739, -75.642, 63.746, 98.133, 16.003]
  MoveL 4470 to (239.85, 154.05, 69.25) mm, rotated rx -180 ry 0 rz 180 deg; joints [-62.601, 57.739, -75.642, 63.746, 98.133, 16.003]
  Call Extruder(262.22712)
  MoveL 4471 to (239.78, 154.27, 69.25) mm, rotated rx -180 ry 0 rz 180 deg; joints [-62.654, 57.752, -75.636, 63.795, 98.109, 15.993]
  MoveL 4472 to (239.78, 154.27, 69.25) mm, rotated rx -180 ry 0 rz 180 deg; joints [-62.654, 57.752, -75.636, 63.795, 98.109, 15.993]
  Call Extruder(262.35848)
  MoveL 4473 to (239.71, 154.49, 69.25) mm, rotated rx -180 ry 0 rz 180 deg; joints [-62.708, 57.766, -75.63, 63.845, 98.086, 15.983]
  MoveL 4474 to (239.71, 154.49, 69.25) mm, rotated rx -180 ry 0 rz 180 deg; joints [-62.708, 57.766, -75.63, 63.845, 98.086, 15.983]
  Call Extruder(262.47038)
  MoveL 4475 to (239.65, 154.68, 69.25) mm, rotated rx 180 ry 0 rz -180 deg; joints [-62.754, 57.777, -75.624, 63.888, 98.066, 15.974]
  MoveL 4476 to (239.65, 154.68, 69.25) mm, rotated rx 180 ry 0 rz -180 deg; joints [-62.754, 57.777, -75.624, 63.888, 98.066, 15.974]
  Call Extruder(262.58272)
  MoveL 4477 to (239.59, 154.87, 69.25) mm, rotated rx -180 ry 0 rz 180 deg; joints [-62.801, 57.788, -75.619, 63.931, 98.046, 15.966]
  MoveL 4478 to (239.59, 154.87, 69.25) mm, rotated rx -180 ry 0 rz 180 deg; joints [-62.801, 57.788, -75.619, 63.931, 98.046, 15.966]
  Call Extruder(262.69551)
  MoveL 4479 to (239.53, 155.06, 69.25) mm, rotated rx -180 ry 0 rz 180 deg; joints [-62.847, 57.799, -75.614, 63.974, 98.026, 15.957]
  MoveL 4480 to (239.53, 155.06, 69.25) mm, rotated rx -180 ry 0 rz 180 deg; joints [-62.847, 57.799, -75.614, 63.974, 98.026, 15.957]
  Call Extruder(262.80875)
  MoveL 4481 to (239.47, 155.25, 69.25) mm, rotated rx -180 ry 0 rz 180 deg; joints [-62.893, 57.81, -75.609, 64.017, 98.006, 15.948]
  MoveL 4482 to (239.47, 155.25, 69.25) mm, rotated rx -180 ry 0 rz 180 deg; joints [-62.893, 57.81, -75.609, 64.017, 98.006, 15.948]
  Call Extruder(262.92243)
  MoveL 4483 to (239.41, 155.44, 69.25) mm, rotated rx -180 ry 0 rz 180 deg; joints [-62.939, 57.821, -75.603, 64.059, 97.986, 15.94]
  MoveL 4484 to (239.41, 155.44, 69.25) mm, rotated rx -180 ry 0 rz 180 deg; joints [-62.939, 57.821, -75.603, 64.059, 97.986, 15.94]
  Call Extruder(263.10439)
  MoveL 4485 to (239.29, 155.73, 69.25) mm, rotated rx 180 ry 0 rz -180 deg; joints [-63.018, 57.837, -75.596, 64.133, 97.954, 15.929]
  MoveL 4486 to (239.29, 155.73, 69.25) mm, rotated rx 180 ry 0 rz -180 deg; joints [-63.018, 57.837, -75.596, 64.133, 97.954, 15.929]
  Call Extruder(263.28710)
  MoveL 4487 to (239.17, 156.02, 69.25) mm, rotated rx -180 ry 0 rz 180 deg; joints [-63.097, 57.854, -75.588, 64.206, 97.922, 15.917]
  MoveL 4488 to (239.17, 156.02, 69.25) mm, rotated rx -180 ry 0 rz 180 deg; joints [-63.097, 57.854, -75.588, 64.206, 97.922, 15.917]
  Call Extruder(263.45752)
  MoveL 4489 to (239.05, 156.29, 69.25) mm, rotated rx 180 ry 0 rz 180 deg; joints [-63.17, 57.869, -75.581, 64.274, 97.892, 15.907]
  MoveL 4490 to (239.05, 156.29, 69.25) mm, rotated rx 180 ry 0 rz 180 deg; joints [-63.17, 57.869, -75.581, 64.274, 97.892, 15.907]
  Call Extruder(263.61554)
  MoveL 4491 to (238.94, 156.54, 69.25) mm, rotated rx 180 ry 0 rz -180 deg; joints [-63.238, 57.882, -75.574, 64.338, 97.865, 15.898]
  MoveL 4492 to (238.94, 156.54, 69.25) mm, rotated rx 180 ry 0 rz -180 deg; joints [-63.238, 57.882, -75.574, 64.338, 97.865, 15.898]
  Call Extruder(263.77415)
  MoveL 4493 to (238.84, 156.79, 69.25) mm, rotated rx -180 ry 0 rz -180 deg; joints [-63.306, 57.896, -75.567, 64.401, 97.838, 15.888]
  MoveL 4494 to (238.84, 156.79, 69.25) mm, rotated rx -180 ry 0 rz -180 deg; joints [-63.306, 57.896, -75.567, 64.401, 97.838, 15.888]
  Call Extruder(263.98032)
  MoveL 4495 to (238.66, 157.09, 69.25) mm, rotated rx 180 ry 0 rz 180 deg; joints [-63.401, 57.911, -75.56, 64.491, 97.802, 15.88]
  MoveL 4496 to (238.66, 157.09, 69.25) mm, rotated rx 180 ry 0 rz 180 deg; joints [-63.401, 57.911, -75.56, 64.491, 97.802, 15.88]
  Call Extruder(264.18727)
  MoveL 4497 to (238.49, 157.4, 69.25) mm, rotated rx -180 ry 0 rz 180 deg; joints [-63.497, 57.927, -75.553, 64.581, 97.766, 15.872]
  MoveL 4498 to (238.49, 157.4, 69.25) mm, rotated rx -180 ry 0 rz 180 deg; joints [-63.497, 57.927, -75.553, 64.581, 97.766, 15.872]
  Call Extruder(264.39499)
  MoveL 4499 to (238.31, 157.7, 69.25) mm, rotated rx -180 ry 0 rz -180 deg; joints [-63.592, 57.942, -75.545, 64.671, 97.73, 15.864]
  MoveL 4500 to (238.31, 157.7, 69.25) mm, rotated rx -180 ry 0 rz -180 deg; joints [-63.592, 57.942, -75.545, 64.671, 97.73, 15.864]
  Call Extruder(264.60350)
  MoveL 4501 to (238.13, 158.01, 69.25) mm, rotated rx -180 ry 0 rz 180 deg; joints [-63.687, 57.957, -75.538, 64.76, 97.694, 15.855]
  MoveL 4502 to (238.13, 158.01, 69.25) mm, rotated rx -180 ry 0 rz 180 deg; joints [-63.687, 57.957, -75.538, 64.76, 97.694, 15.855]
  Call Extruder(264.78304)
  MoveL 4503 to (237.96, 158.25, 69.25) mm, rotated rx 180 ry 0 rz 180 deg; joints [-63.774, 57.969, -75.532, 64.842, 97.664, 15.851]
  MoveL 4504 to (237.96, 158.25, 69.25) mm, rotated rx 180 ry 0 rz 180 deg; joints [-63.774, 57.969, -75.532, 64.842, 97.664, 15.851]
  Call Extruder(265.11645)
  MoveL 4505 to (237.63, 158.7, 69.25) mm, rotated rx -180 ry 0 rz -180 deg; joints [-63.934, 57.989, -75.522, 64.994, 97.607, 15.844]
  MoveL 4506 to (237.63, 158.7, 69.25) mm, rotated rx -180 ry 0 rz -180 deg; joints [-63.934, 57.989, -75.522, 64.994, 97.607, 15.844]
  Call Extruder(265.45104)
  MoveL 4507 to (237.3, 159.15, 69.25) mm, rotated rx 180 ry 0 rz -180 deg; joints [-64.094, 58.01, -75.512, 65.145, 97.55, 15.836]
  Call Extruder(266.27899)
  MoveL 4508 to (236.39, 160.19, 69.25) mm, rotated rx -180 ry 0 rz 180 deg; joints [-64.505, 58.052, -75.491, 65.537, 97.412, 15.83]
  Call Extruder(267.10694)
  MoveL 4509 to (235.35, 161.1, 69.25) mm, rotated rx 180 ry 0 rz -180 deg; joints [-64.933, 58.082, -75.476, 65.947, 97.277, 15.842]
  Call Extruder(267.27424)
  MoveL 4510 to (235.13, 161.27, 69.25) mm, rotated rx -180 ry 0 rz -180 deg; joints [-65.021, 58.086, -75.474, 66.031, 97.25, 15.847]
  MoveL 4511 to (235.13, 161.27, 69.25) mm, rotated rx -180 ry 0 rz -180 deg; joints [-65.021, 58.086, -75.474, 66.031, 97.25, 15.847]
  Call Extruder(267.60766)
  MoveL 4512 to (234.68, 161.59, 69.25) mm, rotated rx 180 ry 0 rz 180 deg; joints [-65.197, 58.095, -75.47, 66.201, 97.197, 15.857]
  MoveL 4513 to (234.68, 161.59, 69.25) mm, rotated rx 180 ry 0 rz 180 deg; joints [-65.197, 58.095, -75.47, 66.201, 97.197, 15.857]
  Call Extruder(267.93990)
  MoveL 4514 to (234.23, 161.92, 69.25) mm, rotated rx 180 ry 0 rz 180 deg; joints [-65.374, 58.103, -75.466, 66.37, 97.143, 15.867]
  MoveL 4515 to (234.23, 161.92, 69.25) mm, rotated rx 180 ry 0 rz 180 deg; joints [-65.374, 58.103, -75.466, 66.37, 97.143, 15.867]
  Call Extruder(268.05756)
  MoveL 4516 to (234.05, 162.02, 69.25) mm, rotated rx -180 ry 0 rz 180 deg; joints [-65.437, 58.105, -75.465, 66.431, 97.125, 15.872]
  MoveL 4517 to (234.05, 162.02, 69.25) mm, rotated rx -180 ry 0 rz 180 deg; joints [-65.437, 58.105, -75.465, 66.431, 97.125, 15.872]
  Call Extruder(268.26529)
  MoveL 4518 to (233.75, 162.2, 69.25) mm, rotated rx 180 ry 0 rz 180 deg; joints [-65.549, 58.107, -75.464, 66.54, 97.093, 15.882]
  MoveL 4519 to (233.75, 162.2, 69.25) mm, rotated rx 180 ry 0 rz 180 deg; joints [-65.549, 58.107, -75.464, 66.54, 97.093, 15.882]
  Call Extruder(268.47224)
  MoveL 4520 to (233.45, 162.37, 69.25) mm, rotated rx -180 ry 0 rz 180 deg; joints [-65.662, 58.11, -75.463, 66.648, 97.061, 15.892]
  MoveL 4521 to (233.45, 162.37, 69.25) mm, rotated rx -180 ry 0 rz 180 deg; joints [-65.662, 58.11, -75.463, 66.648, 97.061, 15.892]
  Call Extruder(268.67841)
  MoveL 4522 to (233.14, 162.55, 69.25) mm, rotated rx 180 ry 0 rz 180 deg; joints [-65.774, 58.113, -75.461, 66.757, 97.028, 15.901]
  MoveL 4523 to (233.14, 162.55, 69.25) mm, rotated rx 180 ry 0 rz 180 deg; joints [-65.774, 58.113, -75.461, 66.757, 97.028, 15.901]
  Call Extruder(268.86008)
  MoveL 4524 to (232.87, 162.69, 69.25) mm, rotated rx -180 ry 0 rz 180 deg; joints [-65.874, 58.114, -75.461, 66.853, 97, 15.911]
  MoveL 4525 to (232.87, 162.69, 69.25) mm, rotated rx -180 ry 0 rz 180 deg; joints [-65.874, 58.114, -75.461, 66.853, 97, 15.911]
  Call Extruder(269.01805)
  MoveL 4526 to (232.62, 162.8, 69.25) mm, rotated rx -180 ry 0 rz 180 deg; joints [-65.961, 58.114, -75.461, 66.938, 96.976, 15.922]
  MoveL 4527 to (232.62, 162.8, 69.25) mm, rotated rx -180 ry 0 rz 180 deg; joints [-65.961, 58.114, -75.461, 66.938, 96.976, 15.922]
  Call Extruder(269.17542)
  MoveL 4528 to (232.37, 162.9, 69.25) mm, rotated rx -180 ry 0 rz 180 deg; joints [-66.048, 58.113, -75.461, 67.022, 96.953, 15.933]
  MoveL 4529 to (232.37, 162.9, 69.25) mm, rotated rx -180 ry 0 rz 180 deg; joints [-66.048, 58.113, -75.461, 67.022, 96.953, 15.933]
  Call Extruder(269.35816)
  MoveL 4530 to (232.07, 163.03, 69.25) mm, rotated rx 180 ry 0 rz -180 deg; joints [-66.149, 58.113, -75.461, 67.12, 96.925, 15.946]
  MoveL 4531 to (232.07, 163.03, 69.25) mm, rotated rx 180 ry 0 rz -180 deg; joints [-66.149, 58.113, -75.461, 67.12, 96.925, 15.946]
  Call Extruder(269.54014)
  MoveL 4532 to (231.78, 163.15, 69.25) mm, rotated rx 180 ry 0 rz -180 deg; joints [-66.251, 58.112, -75.461, 67.219, 96.898, 15.958]
  MoveL 4533 to (231.78, 163.15, 69.25) mm, rotated rx 180 ry 0 rz -180 deg; joints [-66.251, 58.112, -75.461, 67.219, 96.898, 15.958]
  Call Extruder(269.68748)
  MoveL 4534 to (231.54, 163.24, 69.25) mm, rotated rx 180 ry 0 rz -180 deg; joints [-66.333, 58.111, -75.462, 67.299, 96.875, 15.969]
  MoveL 4535 to (231.54, 163.24, 69.25) mm, rotated rx 180 ry 0 rz -180 deg; joints [-66.333, 58.111, -75.462, 67.299, 96.875, 15.969]
  Call Extruder(269.80071)
  MoveL 4536 to (231.35, 163.3, 69.25) mm, rotated rx 180 ry 0 rz -180 deg; joints [-66.397, 58.11, -75.463, 67.361, 96.859, 15.979]
  MoveL 4537 to (231.35, 163.3, 69.25) mm, rotated rx 180 ry 0 rz -180 deg; joints [-66.397, 58.11, -75.463, 67.361, 96.859, 15.979]
  Call Extruder(269.91348)
  MoveL 4538 to (231.17, 163.36, 69.25) mm, rotated rx 180 ry 0 rz 180 deg; joints [-66.46, 58.108, -75.463, 67.422, 96.842, 15.988]
  MoveL 4539 to (231.17, 163.36, 69.25) mm, rotated rx 180 ry 0 rz 180 deg; joints [-66.46, 58.108, -75.463, 67.422, 96.842, 15.988]
  Call Extruder(270.02582)
  MoveL 4540 to (230.98, 163.42, 69.25) mm, rotated rx -180 ry 0 rz 180 deg; joints [-66.524, 58.107, -75.464, 67.484, 96.826, 15.997]
  MoveL 4541 to (230.98, 163.42, 69.25) mm, rotated rx -180 ry 0 rz 180 deg; joints [-66.524, 58.107, -75.464, 67.484, 96.826, 15.997]
  Call Extruder(270.13770)
  MoveL 4542 to (230.79, 163.48, 69.25) mm, rotated rx -180 ry 0 rz 180 deg; joints [-66.587, 58.105, -75.465, 67.545, 96.809, 16.007]
  MoveL 4543 to (230.79, 163.48, 69.25) mm, rotated rx -180 ry 0 rz 180 deg; joints [-66.587, 58.105, -75.465, 67.545, 96.809, 16.007]
  Call Extruder(270.25911)
  MoveL 4544 to (230.58, 163.55, 69.25) mm, rotated rx 180 ry 0 rz -180 deg; joints [-66.656, 58.103, -75.466, 67.613, 96.791, 16.017]
  MoveL 4545 to (230.58, 163.55, 69.25) mm, rotated rx 180 ry 0 rz -180 deg; joints [-66.656, 58.103, -75.466, 67.613, 96.791, 16.017]
  Call Extruder(270.38992)
  MoveL 4546 to (230.36, 163.62, 69.25) mm, rotated rx 180 ry 0 rz 180 deg; joints [-66.731, 58.101, -75.467, 67.685, 96.771, 16.029]
  MoveL 4547 to (230.36, 163.62, 69.25) mm, rotated rx 180 ry 0 rz 180 deg; joints [-66.731, 58.101, -75.467, 67.685, 96.771, 16.029]
  Call Extruder(270.52017)
  MoveL 4548 to (230.14, 163.68, 69.25) mm, rotated rx 180 ry 0 rz 180 deg; joints [-66.805, 58.099, -75.468, 67.758, 96.752, 16.04]
  MoveL 4549 to (230.14, 163.68, 69.25) mm, rotated rx 180 ry 0 rz 180 deg; joints [-66.805, 58.099, -75.468, 67.758, 96.752, 16.04]
  Call Extruder(270.64985)
  MoveL 4550 to (229.91, 163.75, 69.25) mm, rotated rx 180 ry 0 rz -180 deg; joints [-66.88, 58.097, -75.469, 67.831, 96.733, 16.051]
  MoveL 4551 to (229.91, 163.75, 69.25) mm, rotated rx 180 ry 0 rz -180 deg; joints [-66.88, 58.097, -75.469, 67.831, 96.733, 16.051]
  Call Extruder(270.77897)
  MoveL 4552 to (229.69, 163.82, 69.25) mm, rotated rx 180 ry 0 rz 180 deg; joints [-66.955, 58.095, -75.47, 67.903, 96.713, 16.063]
  MoveL 4553 to (229.69, 163.82, 69.25) mm, rotated rx 180 ry 0 rz 180 deg; joints [-66.955, 58.095, -75.47, 67.903, 96.713, 16.063]
  Call Extruder(270.89404)
  MoveL 4554 to (229.48, 163.86, 69.25) mm, rotated rx -180 ry 0 rz 180 deg; joints [-67.021, 58.092, -75.471, 67.968, 96.696, 16.074]
  MoveL 4555 to (229.48, 163.86, 69.25) mm, rotated rx -180 ry 0 rz 180 deg; joints [-67.021, 58.092, -75.471, 67.968, 96.696, 16.074]
  Call Extruder(271.00867)
  MoveL 4556 to (229.28, 163.91, 69.25) mm, rotated rx 180 ry 0 rz 180 deg; joints [-67.087, 58.089, -75.473, 68.032, 96.68, 16.086]
  MoveL 4557 to (229.28, 163.91, 69.25) mm, rotated rx 180 ry 0 rz 180 deg; joints [-67.087, 58.089, -75.473, 68.032, 96.68, 16.086]
  Call Extruder(271.12284)
  MoveL 4558 to (229.08, 163.95, 69.25) mm, rotated rx -180 ry 0 rz 180 deg; joints [-67.153, 58.086, -75.474, 68.097, 96.663, 16.098]
  MoveL 4559 to (229.08, 163.95, 69.25) mm, rotated rx -180 ry 0 rz 180 deg; joints [-67.153, 58.086, -75.474, 68.097, 96.663, 16.098]
  Call Extruder(271.23656)
  MoveL 4560 to (228.87, 164, 69.25) mm, rotated rx -180 ry 0 rz 180 deg; joints [-67.22, 58.083, -75.476, 68.161, 96.646, 16.109]
  MoveL 4561 to (228.87, 164, 69.25) mm, rotated rx -180 ry 0 rz 180 deg; joints [-67.22, 58.083, -75.476, 68.161, 96.646, 16.109]
  Call Extruder(271.36198)
  MoveL 4562 to (228.64, 164.04, 69.25) mm, rotated rx 180 ry 0 rz -180 deg; joints [-67.293, 58.08, -75.478, 68.233, 96.628, 16.122]
  MoveL 4563 to (228.64, 164.04, 69.25) mm, rotated rx 180 ry 0 rz -180 deg; joints [-67.293, 58.08, -75.478, 68.233, 96.628, 16.122]
  Call Extruder(271.49895)
  MoveL 4564 to (228.4, 164.09, 69.25) mm, rotated rx 180 ry 0 rz -180 deg; joints [-67.373, 58.076, -75.48, 68.311, 96.608, 16.137]
  MoveL 4565 to (228.4, 164.09, 69.25) mm, rotated rx 180 ry 0 rz -180 deg; joints [-67.373, 58.076, -75.48, 68.311, 96.608, 16.137]
  Call Extruder(271.63532)
  MoveL 4566 to (228.15, 164.14, 69.25) mm, rotated rx -180 ry 0 rz 180 deg; joints [-67.453, 58.072, -75.482, 68.389, 96.588, 16.151]
  MoveL 4567 to (228.15, 164.14, 69.25) mm, rotated rx -180 ry 0 rz 180 deg; joints [-67.453, 58.072, -75.482, 68.389, 96.588, 16.151]
  Call Extruder(271.77108)
  MoveL 4568 to (227.9, 164.19, 69.25) mm, rotated rx -180 ry 0 rz 180 deg; joints [-67.534, 58.068, -75.483, 68.467, 96.567, 16.165]
  MoveL 4569 to (227.9, 164.19, 69.25) mm, rotated rx -180 ry 0 rz 180 deg; joints [-67.534, 58.068, -75.483, 68.467, 96.567, 16.165]
  Call Extruder(271.90623)
  MoveL 4570 to (227.65, 164.24, 69.25) mm, rotated rx -180 ry 0 rz 180 deg; joints [-67.614, 58.064, -75.485, 68.546, 96.547, 16.18]
  MoveL 4571 to (227.65, 164.24, 69.25) mm, rotated rx -180 ry 0 rz 180 deg; joints [-67.614, 58.064, -75.485, 68.546, 96.547, 16.18]
  Call Extruder(272.04076)
  MoveL 4572 to (227.4, 164.29, 69.25) mm, rotated rx 180 ry 0 rz 180 deg; joints [-67.695, 58.06, -75.487, 68.624, 96.527, 16.194]
  MoveL 4573 to (227.4, 164.29, 69.25) mm, rotated rx 180 ry 0 rz 180 deg; joints [-67.695, 58.06, -75.487, 68.624, 96.527, 16.194]
  Call Extruder(272.17469)
  MoveL 4574 to (227.15, 164.34, 69.25) mm, rotated rx -180 ry 0 rz -180 deg; joints [-67.775, 58.056, -75.489, 68.702, 96.507, 16.208]
  MoveL 4575 to (227.15, 164.34, 69.25) mm, rotated rx -180 ry 0 rz -180 deg; joints [-67.775, 58.056, -75.489, 68.702, 96.507, 16.208]
  Call Extruder(272.32256)
  MoveL 4576 to (226.87, 164.39, 69.25) mm, rotated rx 180 ry 0 rz 180 deg; joints [-67.864, 58.052, -75.491, 68.789, 96.484, 16.224]
  MoveL 4577 to (226.87, 164.39, 69.25) mm, rotated rx 180 ry 0 rz 180 deg; joints [-67.864, 58.052, -75.491, 68.789, 96.484, 16.224]
  Call Extruder(272.48429)
  MoveL 4578 to (226.57, 164.44, 69.25) mm, rotated rx -180 ry 0 rz 180 deg; joints [-67.961, 58.046, -75.494, 68.884, 96.46, 16.243]
  MoveL 4579 to (226.57, 164.44, 69.25) mm, rotated rx -180 ry 0 rz 180 deg; joints [-67.961, 58.046, -75.494, 68.884, 96.46, 16.243]
  Call Extruder(272.64531)
  MoveL 4580 to (226.26, 164.49, 69.25) mm, rotated rx -180 ry 0 rz 180 deg; joints [-68.059, 58.041, -75.497, 68.979, 96.436, 16.261]
  MoveL 4581 to (226.26, 164.49, 69.25) mm, rotated rx -180 ry 0 rz 180 deg; joints [-68.059, 58.041, -75.497, 68.979, 96.436, 16.261]
  Call Extruder(272.80559)
  MoveL 4582 to (225.96, 164.53, 69.25) mm, rotated rx 180 ry 0 rz 180 deg; joints [-68.156, 58.035, -75.5, 69.074, 96.411, 16.279]
  MoveL 4583 to (225.96, 164.53, 69.25) mm, rotated rx 180 ry 0 rz 180 deg; joints [-68.156, 58.035, -75.5, 69.074, 96.411, 16.279]
  Call Extruder(272.96514)
  MoveL 4584 to (225.65, 164.58, 69.25) mm, rotated rx 180 ry 0 rz 180 deg; joints [-68.254, 58.03, -75.502, 69.169, 96.387, 16.297]
  MoveL 4585 to (225.65, 164.58, 69.25) mm, rotated rx 180 ry 0 rz 180 deg; joints [-68.254, 58.03, -75.502, 69.169, 96.387, 16.297]
  Call Extruder(273.12397)
  MoveL 4586 to (225.34, 164.63, 69.25) mm, rotated rx 180 ry 0 rz 180 deg; joints [-68.351, 58.025, -75.505, 69.264, 96.362, 16.315]
  MoveL 4587 to (225.34, 164.63, 69.25) mm, rotated rx 180 ry 0 rz 180 deg; joints [-68.351, 58.025, -75.505, 69.264, 96.362, 16.315]
  Call Extruder(273.30264)
  MoveL 4588 to (225, 164.68, 69.25) mm, rotated rx -180 ry 0 rz 180 deg; joints [-68.461, 58.018, -75.508, 69.372, 96.335, 16.336]
  MoveL 4589 to (225, 164.68, 69.25) mm, rotated rx -180 ry 0 rz 180 deg; joints [-68.461, 58.018, -75.508, 69.372, 96.335, 16.336]
  Call Extruder(273.50108)
  MoveL 4590 to (224.61, 164.73, 69.25) mm, rotated rx -180 ry 0 rz 180 deg; joints [-68.583, 58.01, -75.512, 69.491, 96.304, 16.36]
  MoveL 4591 to (224.61, 164.73, 69.25) mm, rotated rx -180 ry 0 rz 180 deg; joints [-68.583, 58.01, -75.512, 69.491, 96.304, 16.36]
  Call Extruder(273.69866)
  MoveL 4592 to (224.22, 164.77, 69.25) mm, rotated rx 180 ry 0 rz 180 deg; joints [-68.706, 58.003, -75.516, 69.61, 96.274, 16.384]
  MoveL 4593 to (224.22, 164.77, 69.25) mm, rotated rx 180 ry 0 rz 180 deg; joints [-68.706, 58.003, -75.516, 69.61, 96.274, 16.384]
  Call Extruder(273.89536)
  MoveL 4594 to (223.84, 164.82, 69.25) mm, rotated rx 180 ry 0 rz 180 deg; joints [-68.828, 57.995, -75.519, 69.729, 96.243, 16.407]
  MoveL 4595 to (223.84, 164.82, 69.25) mm, rotated rx 180 ry 0 rz 180 deg; joints [-68.828, 57.995, -75.519, 69.729, 96.243, 16.407]
  Call Extruder(274.09120)
  MoveL 4596 to (223.45, 164.86, 69.25) mm, rotated rx -180 ry 0 rz 180 deg; joints [-68.951, 57.987, -75.523, 69.849, 96.213, 16.431]
  MoveL 4597 to (223.45, 164.86, 69.25) mm, rotated rx -180 ry 0 rz 180 deg; joints [-68.951, 57.987, -75.523, 69.849, 96.213, 16.431]
  Call Extruder(274.38656)
  MoveL 4598 to (222.86, 164.91, 69.25) mm, rotated rx -180 ry 0 rz 180 deg; joints [-69.135, 57.974, -75.53, 70.028, 96.167, 16.469]
  MoveL 4599 to (222.86, 164.91, 69.25) mm, rotated rx -180 ry 0 rz 180 deg; joints [-69.135, 57.974, -75.53, 70.028, 96.167, 16.469]
  Call Extruder(274.68059)
  MoveL 4600 to (222.27, 164.96, 69.25) mm, rotated rx 180 ry 0 rz 180 deg; joints [-69.319, 57.961, -75.536, 70.208, 96.122, 16.506]
  MoveL 4601 to (222.27, 164.96, 69.25) mm, rotated rx 180 ry 0 rz 180 deg; joints [-69.319, 57.961, -75.536, 70.208, 96.122, 16.506]
  Call Extruder(274.97329)
  MoveL 4602 to (221.68, 165, 69.25) mm, rotated rx 180 ry 0 rz 180 deg; joints [-69.504, 57.948, -75.542, 70.388, 96.076, 16.543]
  MoveL 4603 to (221.68, 165, 69.25) mm, rotated rx 180 ry 0 rz 180 deg; joints [-69.504, 57.948, -75.542, 70.388, 96.076, 16.543]
  Call Extruder(275.54673)
  MoveL 4604 to (220.52, 165.05, 69.25) mm, rotated rx -180 ry 0 rz 180 deg; joints [-69.864, 57.92, -75.556, 70.739, 95.987, 16.619]
  MoveL 4605 to (220.52, 165.05, 69.25) mm, rotated rx -180 ry 0 rz 180 deg; joints [-69.864, 57.92, -75.556, 70.739, 95.987, 16.619]
  Call Extruder(276.26074)
  MoveL 4606 to (219.06, 165.09, 69.25) mm, rotated rx 180 ry 0 rz -180 deg; joints [-70.315, 57.884, -75.573, 71.179, 95.875, 16.715]
  Call Extruder(393.10748)
  MoveL 4607 to (-19.06, 165.09, 69.25) mm, rotated rx -180 ry 0 rz 180 deg; joints [-137.325, 62.608, -72.096, 136.932, 83.039, 6.463]
  Call Extruder(393.53608)
  MoveL 4608 to (-19.94, 165.07, 69.25) mm, rotated rx -180 ry 0 rz 180 deg; joints [-137.467, 62.646, -72.055, 137.08, 83.08, 6.392]
  MoveL 4609 to (-19.94, 165.07, 69.25) mm, rotated rx -180 ry 0 rz 180 deg; joints [-137.467, 62.646, -72.055, 137.08, 83.08, 6.392]
  Call Extruder(394.10954)
  MoveL 4610 to (-21.1, 165.03, 69.25) mm, rotated rx -180 ry 0 rz 180 deg; joints [-137.659, 62.694, -72.002, 137.28, 83.134, 6.299]
  MoveL 4611 to (-21.1, 165.03, 69.25) mm, rotated rx -180 ry 0 rz 180 deg; joints [-137.659, 62.694, -72.002, 137.28, 83.134, 6.299]
  Call Extruder(394.54383)
  MoveL 4612 to (-21.97, 164.98, 69.25) mm, rotated rx 180 ry 0 rz 180 deg; joints [-137.804, 62.73, -71.962, 137.432, 83.174, 6.23]
  MoveL 4613 to (-21.97, 164.98, 69.25) mm, rotated rx 180 ry 0 rz 180 deg; joints [-137.804, 62.73, -71.962, 137.432, 83.174, 6.23]
  Call Extruder(394.83786)
  MoveL 4614 to (-22.56, 164.93, 69.25) mm, rotated rx -180 ry 0 rz 180 deg; joints [-137.905, 62.754, -71.936, 137.537, 83.2, 6.184]
  MoveL 4615 to (-22.56, 164.93, 69.25) mm, rotated rx -180 ry 0 rz 180 deg; joints [-137.905, 62.754, -71.936, 137.537, 83.2, 6.184]
  Call Extruder(395.13322)
  MoveL 4616 to (-23.15, 164.89, 69.25) mm, rotated rx 180 ry 0 rz 180 deg; joints [-138.004, 62.778, -71.909, 137.641, 83.226, 6.138]
  MoveL 4617 to (-23.15, 164.89, 69.25) mm, rotated rx 180 ry 0 rz 180 deg; joints [-138.004, 62.778, -71.909, 137.641, 83.226, 6.138]
  Call Extruder(395.37944)
  MoveL 4618 to (-23.64, 164.84, 69.25) mm, rotated rx 180 ry 0 rz 180 deg; joints [-138.088, 62.797, -71.888, 137.728, 83.248, 6.101]
  MoveL 4619 to (-23.64, 164.84, 69.25) mm, rotated rx 180 ry 0 rz 180 deg; joints [-138.088, 62.797, -71.888, 137.728, 83.248, 6.101]
  Call Extruder(395.57615)
  MoveL 4620 to (-24.03, 164.79, 69.25) mm, rotated rx 180 ry 0 rz -180 deg; joints [-138.156, 62.812, -71.871, 137.799, 83.264, 6.071]
  MoveL 4621 to (-24.03, 164.79, 69.25) mm, rotated rx 180 ry 0 rz -180 deg; joints [-138.156, 62.812, -71.871, 137.799, 83.264, 6.071]
  Call Extruder(395.77372)
  MoveL 4622 to (-24.42, 164.75, 69.25) mm, rotated rx -180 ry 0 rz 180 deg; joints [-138.224, 62.827, -71.854, 137.869, 83.281, 6.042]
  MoveL 4623 to (-24.42, 164.75, 69.25) mm, rotated rx -180 ry 0 rz 180 deg; joints [-138.224, 62.827, -71.854, 137.869, 83.281, 6.042]
  Call Extruder(395.97216)
  MoveL 4624 to (-24.8, 164.7, 69.25) mm, rotated rx -180 ry 0 rz 180 deg; joints [-138.292, 62.842, -71.837, 137.939, 83.297, 6.012]
  MoveL 4625 to (-24.8, 164.7, 69.25) mm, rotated rx -180 ry 0 rz 180 deg; joints [-138.292, 62.842, -71.837, 137.939, 83.297, 6.012]
  Call Extruder(396.17147)
  MoveL 4626 to (-25.19, 164.66, 69.25) mm, rotated rx -180 ry 0 rz 180 deg; joints [-138.359, 62.857, -71.82, 138.009, 83.314, 5.983]
  MoveL 4627 to (-25.19, 164.66, 69.25) mm, rotated rx -180 ry 0 rz 180 deg; joints [-138.359, 62.857, -71.82, 138.009, 83.314, 5.983]
  Call Extruder(396.33030)
  MoveL 4628 to (-25.5, 164.61, 69.25) mm, rotated rx 180 ry 0 rz 180 deg; joints [-138.415, 62.868, -71.807, 138.067, 83.326, 5.96]
  MoveL 4629 to (-25.5, 164.61, 69.25) mm, rotated rx 180 ry 0 rz 180 deg; joints [-138.415, 62.868, -71.807, 138.067, 83.326, 5.96]
  Call Extruder(396.48986)
  MoveL 4630 to (-25.8, 164.56, 69.25) mm, rotated rx -180 ry 0 rz -180 deg; joints [-138.47, 62.88, -71.794, 138.124, 83.339, 5.937]
  MoveL 4631 to (-25.8, 164.56, 69.25) mm, rotated rx -180 ry 0 rz -180 deg; joints [-138.47, 62.88, -71.794, 138.124, 83.339, 5.937]
  Call Extruder(396.65015)
  MoveL 4632 to (-26.11, 164.51, 69.25) mm, rotated rx -180 ry 0 rz 180 deg; joints [-138.525, 62.891, -71.781, 138.181, 83.351, 5.914]
  MoveL 4633 to (-26.11, 164.51, 69.25) mm, rotated rx -180 ry 0 rz 180 deg; joints [-138.525, 62.891, -71.781, 138.181, 83.351, 5.914]
  Call Extruder(396.81116)
  MoveL 4634 to (-26.41, 164.46, 69.25) mm, rotated rx 180 ry 0 rz 180 deg; joints [-138.58, 62.902, -71.768, 138.238, 83.363, 5.892]
  MoveL 4635 to (-26.41, 164.46, 69.25) mm, rotated rx 180 ry 0 rz 180 deg; joints [-138.58, 62.902, -71.768, 138.238, 83.363, 5.892]
  Call Extruder(396.97291)
  MoveL 4636 to (-26.72, 164.41, 69.25) mm, rotated rx -180 ry 0 rz 180 deg; joints [-138.635, 62.914, -71.755, 138.295, 83.376, 5.869]
  MoveL 4637 to (-26.72, 164.41, 69.25) mm, rotated rx -180 ry 0 rz 180 deg; joints [-138.635, 62.914, -71.755, 138.295, 83.376, 5.869]
  Call Extruder(397.13538)
  MoveL 4638 to (-27.03, 164.37, 69.25) mm, rotated rx 180 ry 0 rz -180 deg; joints [-138.69, 62.925, -71.742, 138.352, 83.389, 5.846]
  MoveL 4639 to (-27.03, 164.37, 69.25) mm, rotated rx 180 ry 0 rz -180 deg; joints [-138.69, 62.925, -71.742, 138.352, 83.389, 5.846]
  Call Extruder(397.26930)
  MoveL 4640 to (-27.27, 164.32, 69.25) mm, rotated rx -180 ry 0 rz 180 deg; joints [-138.736, 62.934, -71.732, 138.4, 83.398, 5.828]
  MoveL 4641 to (-27.27, 164.32, 69.25) mm, rotated rx -180 ry 0 rz 180 deg; joints [-138.736, 62.934, -71.732, 138.4, 83.398, 5.828]
  Call Extruder(397.40384)
  MoveL 4642 to (-27.52, 164.27, 69.25) mm, rotated rx 180 ry 0 rz -180 deg; joints [-138.783, 62.943, -71.721, 138.448, 83.408, 5.81]
  MoveL 4643 to (-27.52, 164.27, 69.25) mm, rotated rx 180 ry 0 rz -180 deg; joints [-138.783, 62.943, -71.721, 138.448, 83.408, 5.81]
  Call Extruder(397.53899)
  MoveL 4644 to (-27.77, 164.22, 69.25) mm, rotated rx 180 ry 0 rz 180 deg; joints [-138.829, 62.952, -71.711, 138.495, 83.417, 5.792]
  MoveL 4645 to (-27.77, 164.22, 69.25) mm, rotated rx 180 ry 0 rz 180 deg; joints [-138.829, 62.952, -71.711, 138.495, 83.417, 5.792]
  Call Extruder(397.67474)
  MoveL 4646 to (-28.02, 164.17, 69.25) mm, rotated rx -180 ry 0 rz 180 deg; joints [-138.875, 62.961, -71.701, 138.543, 83.427, 5.774]
  MoveL 4647 to (-28.02, 164.17, 69.25) mm, rotated rx -180 ry 0 rz 180 deg; joints [-138.875, 62.961, -71.701, 138.543, 83.427, 5.774]
  Call Extruder(397.81111)
  MoveL 4648 to (-28.27, 164.12, 69.25) mm, rotated rx 180 ry 0 rz -180 deg; joints [-138.921, 62.969, -71.691, 138.591, 83.437, 5.756]
  MoveL 4649 to (-28.27, 164.12, 69.25) mm, rotated rx 180 ry 0 rz -180 deg; joints [-138.921, 62.969, -71.691, 138.591, 83.437, 5.756]
  Call Extruder(397.89597)
  MoveL 4650 to (-28.43, 164.09, 69.25) mm, rotated rx -180 ry 0 rz 180 deg; joints [-138.95, 62.975, -71.684, 138.62, 83.443, 5.745]
  Set speed (130.0 mm/s)
  MoveL 4651 to (-31.76, 163.31, 69.25) mm, rotated rx 180 ry 0 rz 180 deg; joints [-139.581, 63.09, -71.549, 139.271, 83.569, 5.508]
  MoveL 4652 to (-31.76, 163.31, 78.65) mm, rotated rx -180 ry 0 rz 180 deg; joints [-139.581, 64.47, -73.506, 139.228, 83.133, 5.887]
  Call Extruder(395.89597)
  Set speed (40.0 mm/s)
  MoveL 4653 to (-31.76, 163.31, 78.65) mm, rotated rx -180 ry 0 rz 180 deg; joints [-139.581, 64.47, -73.506, 139.228, 83.133, 5.887]
  Call Extruder(0.00000)
  Set speed (130.0 mm/s)
  MoveL 4654 to (-31.64, 163.21, 78.65) mm, rotated rx 180 ry 0 rz 180 deg; joints [-139.581, 64.461, -73.517, 139.226, 83.118, 5.9]
  Call Extruder(2.00000)
  Set speed (40.0 mm/s)
  MoveL 4655 to (-31.64, 163.21, 78.65) mm, rotated rx 180 ry 0 rz 180 deg; joints [-139.581, 64.461, -73.517, 139.226, 83.118, 5.9]
  Set speed (30.0 mm/s)
  MoveL 4656 to (-31.64, 163.21, 78.65) mm, rotated rx 180 ry 0 rz 180 deg; joints [-139.581, 64.461, -73.517, 139.226, 83.118, 5.9]
  Call Extruder(2.18198)
  MoveL 4657 to (-31.93, 163.09, 78.65) mm, rotated rx -180 ry 0 rz -180 deg; joints [-139.645, 64.47, -73.507, 139.291, 83.125, 5.88]
  MoveL 4658 to (-31.93, 163.09, 78.65) mm, rotated rx -180 ry 0 rz -180 deg; joints [-139.645, 64.47, -73.507, 139.291, 83.125, 5.88]
  Call Extruder(2.36471)
  MoveL 4659 to (-32.22, 162.97, 78.65) mm, rotated rx 180 ry 0 rz 180 deg; joints [-139.709, 64.478, -73.497, 139.357, 83.132, 5.861]
  MoveL 4660 to (-32.22, 162.97, 78.65) mm, rotated rx 180 ry 0 rz 180 deg; joints [-139.709, 64.478, -73.497, 139.357, 83.132, 5.861]
  Call Extruder(2.53513)
  MoveL 4661 to (-32.49, 162.85, 78.65) mm, rotated rx 180 ry 0 rz 180 deg; joints [-139.768, 64.486, -73.489, 139.418, 83.139, 5.843]
  MoveL 4662 to (-32.49, 162.85, 78.65) mm, rotated rx 180 ry 0 rz 180 deg; joints [-139.768, 64.486, -73.489, 139.418, 83.139, 5.843]
  Call Extruder(2.69310)
  MoveL 4663 to (-32.74, 162.74, 78.65) mm, rotated rx 180 ry 0 rz 180 deg; joints [-139.823, 64.493, -73.48, 139.474, 83.145, 5.826]
  MoveL 4664 to (-32.74, 162.74, 78.65) mm, rotated rx 180 ry 0 rz 180 deg; joints [-139.823, 64.493, -73.48, 139.474, 83.145, 5.826]
  Call Extruder(2.85168)
  MoveL 4665 to (-32.99, 162.64, 78.65) mm, rotated rx -180 ry 0 rz 180 deg; joints [-139.878, 64.5, -73.472, 139.53, 83.151, 5.81]
  MoveL 4666 to (-32.99, 162.64, 78.65) mm, rotated rx -180 ry 0 rz 180 deg; joints [-139.878, 64.5, -73.472, 139.53, 83.151, 5.81]
  Call Extruder(3.05784)
  MoveL 4667 to (-33.29, 162.46, 78.65) mm, rotated rx -180 ry 0 rz 180 deg; joints [-139.953, 64.507, -73.464, 139.607, 83.155, 5.791]
  MoveL 4668 to (-33.29, 162.46, 78.65) mm, rotated rx -180 ry 0 rz 180 deg; joints [-139.953, 64.507, -73.464, 139.607, 83.155, 5.791]
  Call Extruder(3.26479)
  MoveL 4669 to (-33.6, 162.29, 78.65) mm, rotated rx -180 ry 0 rz 180 deg; joints [-140.028, 64.514, -73.456, 139.683, 83.158, 5.772]
  MoveL 4670 to (-33.6, 162.29, 78.65) mm, rotated rx -180 ry 0 rz 180 deg; joints [-140.028, 64.514, -73.456, 139.683, 83.158, 5.772]
  Call Extruder(3.47251)
  MoveL 4671 to (-33.9, 162.11, 78.65) mm, rotated rx 180 ry 0 rz -180 deg; joints [-140.103, 64.52, -73.448, 139.759, 83.162, 5.754]
  MoveL 4672 to (-33.9, 162.11, 78.65) mm, rotated rx 180 ry 0 rz -180 deg; joints [-140.103, 64.52, -73.448, 139.759, 83.162, 5.754]
  Call Extruder(3.68102)
  MoveL 4673 to (-34.21, 161.93, 78.65) mm, rotated rx -180 ry 0 rz 180 deg; joints [-140.178, 64.527, -73.44, 139.835, 83.166, 5.735]
  MoveL 4674 to (-34.21, 161.93, 78.65) mm, rotated rx -180 ry 0 rz 180 deg; joints [-140.178, 64.527, -73.44, 139.835, 83.166, 5.735]
  Call Extruder(3.86055)
  MoveL 4675 to (-34.45, 161.76, 78.65) mm, rotated rx -180 ry 0 rz 180 deg; joints [-140.244, 64.532, -73.435, 139.902, 83.167, 5.721]
  MoveL 4676 to (-34.45, 161.76, 78.65) mm, rotated rx -180 ry 0 rz 180 deg; joints [-140.244, 64.532, -73.435, 139.902, 83.167, 5.721]
  Call Extruder(4.19399)
  MoveL 4677 to (-34.9, 161.43, 78.65) mm, rotated rx -180 ry 0 rz 180 deg; joints [-140.366, 64.54, -73.425, 140.026, 83.168, 5.695]
  MoveL 4678 to (-34.9, 161.43, 78.65) mm, rotated rx -180 ry 0 rz 180 deg; joints [-140.366, 64.54, -73.425, 140.026, 83.168, 5.695]
  Call Extruder(4.52861)
  MoveL 4679 to (-35.35, 161.1, 78.65) mm, rotated rx -180 ry 0 rz 180 deg; joints [-140.489, 64.548, -73.416, 140.15, 83.169, 5.669]
  Call Extruder(5.35652)
  MoveL 4680 to (-36.39, 160.19, 78.65) mm, rotated rx -180 ry 0 rz 180 deg; joints [-140.797, 64.561, -73.401, 140.461, 83.16, 5.614]
  Call Extruder(6.18445)
  MoveL 4681 to (-37.3, 159.15, 78.65) mm, rotated rx -180 ry 0 rz 180 deg; joints [-141.109, 64.564, -73.397, 140.774, 83.135, 5.573]
  Call Extruder(6.35176)
  MoveL 4682 to (-37.47, 158.93, 78.65) mm, rotated rx -180 ry 0 rz 180 deg; joints [-141.172, 64.563, -73.398, 140.837, 83.128, 5.566]
  MoveL 4683 to (-37.47, 158.93, 78.65) mm, rotated rx -180 ry 0 rz 180 deg; joints [-141.172, 64.563, -73.398, 140.837, 83.128, 5.566]
  Call Extruder(6.68519)
  MoveL 4684 to (-37.79, 158.48, 78.65) mm, rotated rx -180 ry 0 rz 180 deg; joints [-141.298, 64.561, -73.4, 140.963, 83.113, 5.553]
  MoveL 4685 to (-37.79, 158.48, 78.65) mm, rotated rx -180 ry 0 rz 180 deg; joints [-141.298, 64.561, -73.4, 140.963, 83.113, 5.553]
  Call Extruder(7.01743)
  MoveL 4686 to (-38.12, 158.03, 78.65) mm, rotated rx 180 ry 0 rz 180 deg; joints [-141.424, 64.56, -73.402, 141.09, 83.098, 5.54]
  MoveL 4687 to (-38.12, 158.03, 78.65) mm, rotated rx 180 ry 0 rz 180 deg; joints [-141.424, 64.56, -73.402, 141.09, 83.098, 5.54]
  Call Extruder(7.13511)
  MoveL 4688 to (-38.22, 157.85, 78.65) mm, rotated rx 180 ry 0 rz 180 deg; joints [-141.468, 64.558, -73.404, 141.134, 83.091, 5.537]
  MoveL 4689 to (-38.22, 157.85, 78.65) mm, rotated rx 180 ry 0 rz 180 deg; joints [-141.468, 64.558, -73.404, 141.134, 83.091, 5.537]
  Call Extruder(7.34283)
  MoveL 4690 to (-38.4, 157.55, 78.65) mm, rotated rx -180 ry 0 rz 180 deg; joints [-141.547, 64.555, -73.407, 141.212, 83.079, 5.532]
  MoveL 4691 to (-38.4, 157.55, 78.65) mm, rotated rx -180 ry 0 rz 180 deg; joints [-141.547, 64.555, -73.407, 141.212, 83.079, 5.532]
  Call Extruder(7.54978)
  MoveL 4692 to (-38.57, 157.25, 78.65) mm, rotated rx -180 ry 0 rz 180 deg; joints [-141.625, 64.552, -73.411, 141.29, 83.066, 5.526]
  MoveL 4693 to (-38.57, 157.25, 78.65) mm, rotated rx -180 ry 0 rz 180 deg; joints [-141.625, 64.552, -73.411, 141.29, 83.066, 5.526]
  Call Extruder(7.75595)
  MoveL 4694 to (-38.75, 156.94, 78.65) mm, rotated rx 180 ry 0 rz -180 deg; joints [-141.704, 64.549, -73.414, 141.368, 83.054, 5.521]
  MoveL 4695 to (-38.75, 156.94, 78.65) mm, rotated rx 180 ry 0 rz -180 deg; joints [-141.704, 64.549, -73.414, 141.368, 83.054, 5.521]
  Call Extruder(7.93762)
  MoveL 4696 to (-38.89, 156.67, 78.65) mm, rotated rx 180 ry 0 rz -180 deg; joints [-141.773, 64.546, -73.418, 141.437, 83.041, 5.517]
  MoveL 4697 to (-38.89, 156.67, 78.65) mm, rotated rx 180 ry 0 rz -180 deg; joints [-141.773, 64.546, -73.418, 141.437, 83.041, 5.517]
  Call Extruder(8.09561)
  MoveL 4698 to (-39, 156.42, 78.65) mm, rotated rx 180 ry 0 rz 180 deg; joints [-141.832, 64.542, -73.423, 141.496, 83.029, 5.515]
  MoveL 4699 to (-39, 156.42, 78.65) mm, rotated rx 180 ry 0 rz 180 deg; joints [-141.832, 64.542, -73.423, 141.496, 83.029, 5.515]
